# B&R Automation Studio project AutomatedPongGame
Automation Studio 4.12.6.106; technology packages: Acp10Arnc0 5.30.2, mappView 5.16.1

## Configuration AutomatedPongGame_UnitTests

CPU 4PPC70.0573-20B, AutomationRuntime R4.93, Build 4.1.2

### Task classes (Cpu.sw)
```
Cyclic#4 (cycle 10000 us):
  Tests_Incl <- UnitTests.UnitTests.Tests_InclinoSensor_C.prg
  Tests_Padd <- UnitTests.UnitTests.Tests_PaddleMotor_C.prg
  Tests_Fiel <- UnitTests.UnitTests.Tests_FieldMotor_C.prg
  Tests_Pong <- UnitTests.UnitTests.Tests_PongGame_C.prg
  Tests_Ball <- UnitTests.UnitTests.Tests_BallControl_C.prg
  Tests_Fie1 <- UnitTests.UnitTests.Tests_FieldControl_C.prg
  Tests_Dist <- UnitTests.UnitTests.Tests_DistanceSensor_C.prg
  Tests_Shoo <- UnitTests.UnitTests.Tests_Shooter_C.prg
Binaries: mvLoader, udbdef, TCData, iomap, asfw, arconfig, ashwd, sysconf, ashwac
Libraries: Runtime, sys_lib, AsIecCon, astime, AsARCfg, AsBrStr, UnitTest, UtWs, UtMgr, Library, arssl, fileio, standard
```

### Hardware
```
4PPC70_0573_20B : 4PPC70.0573-20B v1.6.1.0
  Connector IF2:
    ActivateDevice = 1
    InaPort = 11160
  ConfigurationID = AutomatedPongGame_TS_UnitTest_Sample
  Cyclic4Duration = 10000
  FileDevice1
  FileDeviceName1 = USER
  FileDevicePath1 = USER_PATH
  ActivateDtmServer = 1
  ActivateOpcUa = 1
  OpcUaInformationModels_PV_Version = 1
  KeyMappingFile = VC\4PPC70_0573_20B.dis
```

## Configuration AutomatedPongGame_config

CPU 4PPC70.0573-20B, AutomationRuntime R4.93, Build 4.1.2, Safety 0.0, Vc V4.73.4

### Task classes (Cpu.sw)
```
Cyclic#1 (cycle 2000 us, tolerance 0 us):
  gAxis01Bas <- gAxis01obj.gAxis01Basic.prg
  gAxis02Bas <- gAxis02obj.gAxis02Basic.prg
  Main <- Main.prg
NcDataObjects: acp10etxen <- acp10etxen.dob, gAxis01a <- gAxis01obj.gAxis01a.dob, gAxis01i <- gAxis01obj.gAxis01i.dob, gAxis02a <- gAxis02obj.gAxis02a.dob, gAxis02i <- gAxis02obj.gAxis02i.dob
VcDataObjects: Visu <- Visu.dob
Binaries: udbdef, FWRules, TCData, mvLoader, vcctext, arialbd, vcpdi855, vcdsloc, vcbclass, vcfntttf, Visu03, vcshared, vcrt, vcpk, vcfile, vccbtn, vcmgr, vctcal, vcptelo, vcalarm, vccnum, vcpdsw, Visu01, vcgclass, vcpdihd, vcpdi815, vcpfppc7, vcdsint, Visu02, calibrib, vccbmp, arial, vccstr, Acp10map, acp10cfg, iomap, ashwac, Role, sysconf, arconfig, asfw, User, ashwd, asnxdb1, User_1
Libraries: standard, sys_lib, brsystem, runtime, AsBrStr, Acp10man, Acp10par, NcGlobal, Acp10sdc, Acp10_MC, Library, arssl, astime, powerlnk, fileio, vcresman, AsARCfg, DataObj
```

### Hardware
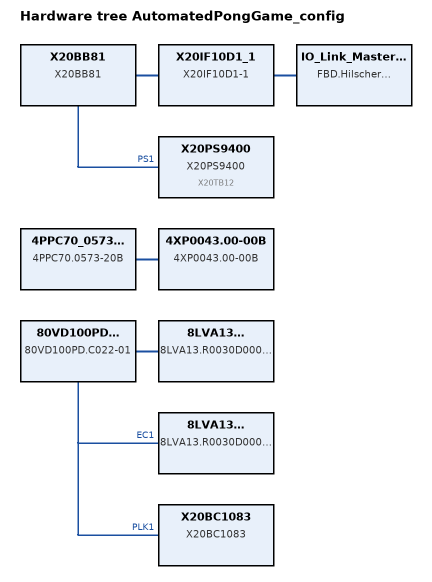
```
4PPC70_0573_20B : 4PPC70.0573-20B v1.6.1.0
  Connector IF1:
    InternetAddress = 192.168.30.1
    SubnetMask = 255.255.255.0
    ActivateIna = 1
  Connector IF2:
    ActivateDevice = 1
    Mode = Manual
    InternetAddress = 192.168.1.20
    SubnetMask = 255.255.255.0
    InaNodeNumber = 0
    Vnc1
    VncAuthentication1 = 1
    VncPasswordViewOnly1 = user
    VncPasswordViewControl1 = admin
    ActivateSnmp = 2
  ConfigurationID = AutomatedPongGame_Config1
  PermanentPvSize = 108
  RemanentGlobalPvSize = 108
  TimerDeviceType = EPLX2X
  TimerDevice = 4PPC70_0573_20B.IF1
  TaskClassIdleTime = 2000
  Cyclic1Duration = 2000
  Cyclic1Tolerance = 0
  Cyclic1Output = 1
  FileDevice1
  FileDeviceName1 = USER
  FileDevicePath1 = USER_PATH
  ActivateDtmServer = 1
  ActivateOpcUa = 1
  OpcUaInformationModels_PV_Version = 1
  VcObjectName = Visu
  KeyMappingFile = VC\4PPC70_0573_20B.dis
4XP0043.00-00B : 4XP0043.00-00B v2.1.1.0  [X2X1 -> 4PPC70_0573_20B.IF5 [Cable Type=X2XCable, Length=10, Version=1.0.0.3]]
80VD100PD.C022-01 : 80VD100PD.C022-01 v2.5.0.0  [PLK1 -> X20BC1083.PLK1 (NodeNumber=2) [Cable Type=PowerlinkCable, Length=10, Version=1.0.0.3]; EC1 -> 8LVA13.R0030D000-0a.EC; EC2 -> 8LVA13.R0030D000-0.EC; MT2 -> 8LVA13.R0030D000-0.MT]
  MotionTP = Acp10Arnc0
  BothEndSwitchesAreNormallyOpen_r1 = on
  QuickStopIsNormallyOpen_r1 = on
  BothEndSwitchesAreNormallyOpen_r2 = on
  QuickStopIsNormallyOpen_r2 = on
8LVA13.R0030D000-0 : 8LVA13.R0030D000-0 v2.2.0.5  [EC -> 80VD100PD.C022-01.EC2; MT -> 80VD100PD.C022-01.MT2]
8LVA13.R0030D000-0a : 8LVA13.R0030D000-0 v2.2.0.5  [EC -> 80VD100PD.C022-01.EC1; MT -> 80VD100PD.C022-01.MT1]
IO_Link_Master_SL_EIP_8P_IP67_V1_5 : FBD.Hilscher.EIGenEDSAdapterDTM.IO-Link Master SL EIP 8P IP67 V1.5 v1.5 (OrderNumber=IO-Link Master SL EIP 8P IP67 V1.5, VendorAddress=192.168.1.150)  [EIP1 -> X20IF10D1_1.IF1]
  DtmId = cae6d7b0-cfd8-47f1-9e8e-3783e9b887dc
  ChannelBlocks_78e66418-9731-44dc-bd45-61a937da4e16  // Module 0
  IO_InputImage_78e66418-9731-44dc-bd45-61a937da4e16  // 446 Byte(s)
  IO_OutputImage_78e66418-9731-44dc-bd45-61a937da4e16  // 302 Byte(s)
X20BB81 : X20BB81 v1.2.0.0
X20BC1083 : X20BC1083 v2.17.0.0  [PLK1 -> 80VD100PD.C022-01.PLK1 (NodeNumber=1) [Cable Type=PowerlinkCable, Length=10, Version=1.0.0.3]; PLK2 -> 4PPC70_0573_20B.IF1 (NodeNumber=1) [Cable Type=PowerlinkCable, Length=10, Version=1.0.0.3]; SL -> X20BB81.SL1]
X20IF10D1_1 : X20IF10D1-1 v1.7.0.0  [SS -> X20BB81.SS1]
  Connector IF1:
    DtmId = 66a43618-f239-4c0c-80e6-69720443d023
  ConfigFile = X20IF10D1_1.dtm
  ConfigModule = asnxdb1
  CycleTime = 2000
X20PS9400 : X20PS9400 v1.9.0.0  [SS1 -> X20TB12.SS; PS -> X20BB81.PS1]
X20TB12 : X20TB12 v1.0.0.0
```

### IoMap.iom - 4PPC70_0573_20B/IoMap.iom
```iecst
VAR_CONFIG
	::digitalInput AT %IB."IO_Link_Master_SL_EIP_8P_IP67_V1_5".Module_0_Input001;
	::gAxis01Bas:BasicControl.Command.MoveJogNeg AT %QX."4XP0043.00-00B".DigitalOutput03;
	::g_Shooter.IO.Shoot AT %QX."4XP0043.00-00B".DigitalOutput07;
	::digitalOutput AT %QB."IO_Link_Master_SL_EIP_8P_IP67_V1_5".Module_0_Output001;
	::g_PaddleMotor.HMI.MoveJogNeg AT %IX."4XP0043.00-00B".DigitalInput01;
	::g_Shooter.HMI.Shoot AT %IX."4XP0043.00-00B".DigitalInput02;
	::g_PaddleMotor.HMI.MoveJogPos AT %IX."4XP0043.00-00B".DigitalInput03;
	::g_DistanceSensorLeft.IO.DataMSB AT %IB."IO_Link_Master_SL_EIP_8P_IP67_V1_5".Module_0_Input415;
	::g_DistanceSensorLeft.IO.DataLSB AT %IB."IO_Link_Master_SL_EIP_8P_IP67_V1_5".Module_0_Input416;
	::g_DistanceSensorRight.IO.DataMSB AT %IB."IO_Link_Master_SL_EIP_8P_IP67_V1_5".Module_0_Input383;
	::g_DistanceSensorRight.IO.DataLSB AT %IB."IO_Link_Master_SL_EIP_8P_IP67_V1_5".Module_0_Input384;
	::g_DistanceSensorMiddle.IO.DataMSB AT %IB."IO_Link_Master_SL_EIP_8P_IP67_V1_5".Module_0_Input351;
	::g_DistanceSensorMiddle.IO.DataLSB AT %IB."IO_Link_Master_SL_EIP_8P_IP67_V1_5".Module_0_Input352;
	::gAxis01Bas:BasicControl.Command.MoveJogPos AT %QX."4XP0043.00-00B".DigitalOutput11;
	::g_InclinoSensor.IO.DataMSB AT %IB."IO_Link_Master_SL_EIP_8P_IP67_V1_5".Module_0_Input319;
	::g_InclinoSensor.IO.DataLSB AT %IB."IO_Link_Master_SL_EIP_8P_IP67_V1_5".Module_0_Input320;
	::g_DistanceSensorMiddle.IO.SensorInfo AT %IB."IO_Link_Master_SL_EIP_8P_IP67_V1_5".Module_0_Input358;
	::g_DistanceSensorRight.IO.SensorInfo AT %IB."IO_Link_Master_SL_EIP_8P_IP67_V1_5".Module_0_Input390;
	::g_DistanceSensorLeft.IO.SensorInfo AT %IB."IO_Link_Master_SL_EIP_8P_IP67_V1_5".Module_0_Input422;
	::g_InclinoSensor.IO.SetCenterPoint AT %QB."IO_Link_Master_SL_EIP_8P_IP67_V1_5".Module_0_Output175;
END_VAR
```

## Configuration Config1

CPU 4PPC70.0573-20B, AutomationRuntime R4.93, Build 4.1.2, Safety 0.0, Vc V4.73.4

### Task classes (Cpu.sw)
```
Cyclic#1 (cycle 2000 us, tolerance 0 us):
  gAxis01Bas <- gAxis01obj.gAxis01Basic.prg
  gAxis02Bas <- gAxis02obj.gAxis02Basic.prg
  Main <- Main.prg
Cyclic#4:
  TonTimer <- Timer_CPP.TonTimer.prg
NcDataObjects: acp10etxen <- acp10etxen.dob, gAxis01a <- gAxis01obj.gAxis01a.dob, gAxis01i <- gAxis01obj.gAxis01i.dob, gAxis02a <- gAxis02obj.gAxis02a.dob, gAxis02i <- gAxis02obj.gAxis02i.dob
VcDataObjects: Visu <- Visu.dob
Binaries: udbdef, FWRules, TCData, mvLoader, vcctext, arialbd, vcpdi855, vcdsloc, vcbclass, vcfntttf, Visu03, vcshared, vcrt, vcpk, vcfile, vccbtn, vcmgr, vctcal, vcptelo, vcalarm, vccnum, vcpdsw, Visu01, vcgclass, vcpdihd, vcpdi815, vcpfppc7, vcdsint, Visu02, calibrib, vccbmp, arial, vccstr, Acp10map, acp10cfg, iomap, ashwac, Role, sysconf, arconfig, asfw, User, ashwd, asnxdb1, User_1
Libraries: Timer, standard, sys_lib, brsystem, runtime, AsBrStr, Acp10man, Acp10par, NcGlobal, Acp10sdc, Acp10_MC, Library, arssl, astime, powerlnk, fileio, dataobj, vcresman
```

### Hardware
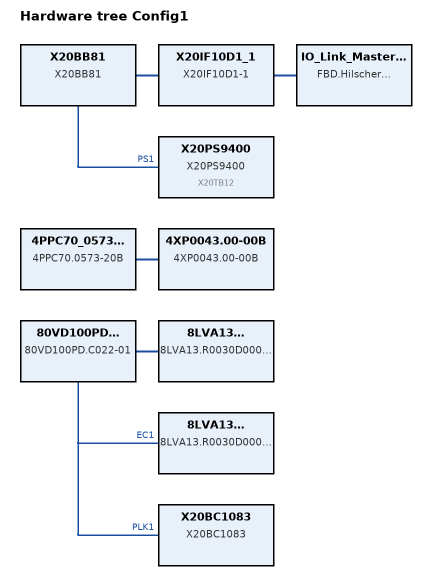
```
4PPC70_0573_20B : 4PPC70.0573-20B v1.6.1.0
  Connector IF1:
    InternetAddress = 192.168.30.1
    SubnetMask = 255.255.255.0
    ActivateIna = 1
  Connector IF2:
    ActivateDevice = 1
    Mode = Manual
    InternetAddress = 192.168.1.20
    SubnetMask = 255.255.255.0
    InaNodeNumber = 0
    Vnc1
    VncAuthentication1 = 1
    VncPasswordViewOnly1 = user
    VncPasswordViewControl1 = admin
    ActivateSnmp = 2
  ConfigurationID = AutomatedPongGame_Config1
  TimerDeviceType = EPLX2X
  TimerDevice = 4PPC70_0573_20B.IF1
  TaskClassIdleTime = 2000
  Cyclic1Duration = 2000
  Cyclic1Tolerance = 0
  Cyclic1Output = 1
  FileDevice1
  FileDeviceName1 = USER
  FileDevicePath1 = USER_PATH
  ActivateDtmServer = 1
  ActivateOpcUa = 1
  OpcUaInformationModels_PV_Version = 1
  VcObjectName = Visu
  KeyMappingFile = VC\4PPC70_0573_20B.dis
4XP0043.00-00B : 4XP0043.00-00B v2.1.1.0  [X2X1 -> 4PPC70_0573_20B.IF5 [Cable Type=X2XCable, Length=10, Version=1.0.0.3]]
80VD100PD.C022-01 : 80VD100PD.C022-01 v2.5.0.0  [PLK1 -> X20BC1083.PLK1 (NodeNumber=2) [Cable Type=PowerlinkCable, Length=10, Version=1.0.0.3]; EC1 -> 8LVA13.R0030D000-0a.EC; EC2 -> 8LVA13.R0030D000-0.EC; MT2 -> 8LVA13.R0030D000-0.MT]
  MotionTP = Acp10Arnc0
  BothEndSwitchesAreNormallyOpen_r1 = on
  QuickStopIsNormallyOpen_r1 = on
  BothEndSwitchesAreNormallyOpen_r2 = on
  QuickStopIsNormallyOpen_r2 = on
8LVA13.R0030D000-0 : 8LVA13.R0030D000-0 v2.2.0.5  [EC -> 80VD100PD.C022-01.EC2; MT -> 80VD100PD.C022-01.MT2]
8LVA13.R0030D000-0a : 8LVA13.R0030D000-0 v2.2.0.5  [EC -> 80VD100PD.C022-01.EC1; MT -> 80VD100PD.C022-01.MT1]
IO_Link_Master_SL_EIP_8P_IP67_V1_5 : FBD.Hilscher.EIGenEDSAdapterDTM.IO-Link Master SL EIP 8P IP67 V1.5 v1.5 (OrderNumber=IO-Link Master SL EIP 8P IP67 V1.5, VendorAddress=192.168.1.150)  [EIP1 -> X20IF10D1_1.IF1]
  DtmId = cae6d7b0-cfd8-47f1-9e8e-3783e9b887dc
  ChannelBlocks_78e66418-9731-44dc-bd45-61a937da4e16  // Module 0
  IO_InputImage_78e66418-9731-44dc-bd45-61a937da4e16  // 446 Byte(s)
  IO_OutputImage_78e66418-9731-44dc-bd45-61a937da4e16  // 302 Byte(s)
X20BB81 : X20BB81 v1.2.0.0
X20BC1083 : X20BC1083 v2.17.0.0  [PLK1 -> 80VD100PD.C022-01.PLK1 (NodeNumber=1) [Cable Type=PowerlinkCable, Length=10, Version=1.0.0.3]; PLK2 -> 4PPC70_0573_20B.IF1 (NodeNumber=1) [Cable Type=PowerlinkCable, Length=10, Version=1.0.0.3]; SL -> X20BB81.SL1]
X20IF10D1_1 : X20IF10D1-1 v1.7.0.0  [SS -> X20BB81.SS1]
  Connector IF1:
    DtmId = 66a43618-f239-4c0c-80e6-69720443d023
  ConfigFile = X20IF10D1_1.dtm
  ConfigModule = asnxdb1
  CycleTime = 2000
X20PS9400 : X20PS9400 v1.9.0.0  [SS1 -> X20TB12.SS; PS -> X20BB81.PS1]
X20TB12 : X20TB12 v1.0.0.0
```

### IoMap.iom - 4PPC70_0573_20B/IoMap.iom
```iecst
VAR_CONFIG
	::digitalInput AT %IB."IO_Link_Master_SL_EIP_8P_IP67_V1_5".Module_0_Input001;
	::gAxis01Bas:BasicControl.Command.MoveJogNeg AT %QX."4XP0043.00-00B".DigitalOutput03;
	::g_Shooter.IO.Shoot AT %QX."4XP0043.00-00B".DigitalOutput07;
	::digitalOutput AT %QB."IO_Link_Master_SL_EIP_8P_IP67_V1_5".Module_0_Output001;
	::g_PaddleMotor.HMI.MoveJogNeg AT %IX."4XP0043.00-00B".DigitalInput01;
	::g_Shooter.HMI.Shoot AT %IX."4XP0043.00-00B".DigitalInput02;
	::g_PaddleMotor.HMI.MoveJogPos AT %IX."4XP0043.00-00B".DigitalInput03;
	::g_DistanceSensorLeft.IO.DataMSB AT %IB."IO_Link_Master_SL_EIP_8P_IP67_V1_5".Module_0_Input415;
	::g_DistanceSensorLeft.IO.DataLSB AT %IB."IO_Link_Master_SL_EIP_8P_IP67_V1_5".Module_0_Input416;
	::g_DistanceSensorRight.IO.DataMSB AT %IB."IO_Link_Master_SL_EIP_8P_IP67_V1_5".Module_0_Input383;
	::g_DistanceSensorRight.IO.DataLSB AT %IB."IO_Link_Master_SL_EIP_8P_IP67_V1_5".Module_0_Input384;
	::g_DistanceSensorMiddle.IO.DataMSB AT %IB."IO_Link_Master_SL_EIP_8P_IP67_V1_5".Module_0_Input351;
	::g_DistanceSensorMiddle.IO.DataLSB AT %IB."IO_Link_Master_SL_EIP_8P_IP67_V1_5".Module_0_Input352;
	::gAxis01Bas:BasicControl.Command.MoveJogPos AT %QX."4XP0043.00-00B".DigitalOutput11;
	::g_InclinoSensor.IO.DataMSB AT %IB."IO_Link_Master_SL_EIP_8P_IP67_V1_5".Module_0_Input319;
	::g_InclinoSensor.IO.DataLSB AT %IB."IO_Link_Master_SL_EIP_8P_IP67_V1_5".Module_0_Input320;
	::g_DistanceSensorMiddle.IO.SensorInfo AT %IB."IO_Link_Master_SL_EIP_8P_IP67_V1_5".Module_0_Input358;
	::g_DistanceSensorRight.IO.SensorInfo AT %IB."IO_Link_Master_SL_EIP_8P_IP67_V1_5".Module_0_Input390;
	::g_DistanceSensorLeft.IO.SensorInfo AT %IB."IO_Link_Master_SL_EIP_8P_IP67_V1_5".Module_0_Input422;
END_VAR
```

### Acp10cfg.ncc - 4PPC70_0573_20B/Motion/Acp10cfg.ncc
```
NcConfiguration (Version=5.30.2, NcSwId=Acp10)
  ACP10CF1_typ:
    cnt_nettrc_rec_drive = 1500
    bufsize_trace_upload = 1200
    tc_nc_man_task = Cyclic #1
    glob_pv_as_ncobject = Yes
    ncsys_dl_broadcast = Yes
    ncsys_dl_acp_reset = Yes
    safemc_log_err_to_ax = Yes
    network_init:
      ncsw_init_execute = Yes
      automatic_execute = No
      node_nr_warning = Yes
      net_err_before_ncact = Yes
    nettrc:
      enter_parsecrec = Yes
      enter_ncaction = Yes
      save_ring_startidx = Yes
    cam_prof_download:
      cam_dat_dl_parallel = No
      tc_cam_dl_parallel = Task class for NC Manager task
    plk_if[0]:
      if_name = IF1
      tc_CycDat_PLCopen = Task class for NC Manager task
      mc_broadcast_extdat = No
```

### Acp10map.ncm - 4PPC70_0573_20B/Motion/Acp10map.ncm
```
NcMapping (NcSwId=Acp10)
  NcObject gAxis01 (ModuleId=80VD100PD.C022-01, Type=ncAXIS, Channel=1, AcoposSimulation=Off, InitParameter=gAxis01i, AcoposParameter=gAxis01a, Disabled=FALSE, ModuleDisabled=FALSE)
  NcObject gAxis02 (ModuleId=80VD100PD.C022-01, Type=ncAXIS, Channel=2, AcoposSimulation=Off, InitParameter=gAxis02i, AcoposParameter=gAxis02a, Disabled=FALSE, ModuleDisabled=FALSE)
  NcObject 80VD100PD.C022-01_ncV_AXIS1 (ModuleId=80VD100PD.C022-01, Type=ncV_AXIS, Channel=1, Disabled=TRUE, ModuleDisabled=FALSE)
  NcObject 80VD100PD.C022-01_ncV_AXIS2 (ModuleId=80VD100PD.C022-01, Type=ncV_AXIS, Channel=2, Disabled=TRUE, ModuleDisabled=FALSE)
```

## Configuration TS_UnitTest_Sample

### Task classes (Cpu.sw)
```
Cyclic#4 (cycle 10000 us):
  SPL_CalcTe <- UnitTestSample.Samples.Tests_Program.Tests_MyCalcLib_C.SPL_CalcTest.prg
  SPL_CalcT1 <- UnitTestSample.Samples.Tests_Program.Tests_MyCalcLib_C.SPL_CalcTest_Variants.prg
  Tests_Padd <- UnitTests.HelperTool_Supported.Tests_PaddleMotor_C.prg
Binaries: mvLoader, udbdef, TCData, iomap, asfw, arconfig, ashwd, sysconf, ashwac
Libraries: Runtime, sys_lib, AsIecCon, astime, AsARCfg, AsBrStr, UnitTest, UtWs, UtMgr, SPLMyCalc, Library, arssl, fileio
```

### Hardware
```
4PPC70_0573_20B : 4PPC70.0573-20B v1.6.1.0
  Connector IF2:
    ActivateDevice = 1
    InaPort = 11160
  ConfigurationID = AutomatedPongGame_TS_UnitTest_Sample
  Cyclic4Duration = 10000
  FileDevice1
  FileDeviceName1 = USER
  FileDevicePath1 = USER_PATH
  KeyMappingFile = VC\4PPC70_0573_20B.dis
```

## Logical view

Binary libraries used (declarations not repeated): UtMgr 2.02.0, UtWs 2.02.0, operator, runtime, astime, AsIecCon, standard, sys_lib, brsystem, AsBrStr, Acp10man 5.30.2, Acp10par 5.30.2, NcGlobal 5.30.2, Acp10sdc 5.30.2, Acp10_MC 5.30.2, AsARCfg, DataObj

### Global.var - Global variables
```iecst
VAR
	gAxis01 : ACP10AXIS_typ;
	gAxis02 : ACP10AXIS_typ;
	digitalInput : USINT;
	g_PongGame : UDT_PongGame := (ALM:=(PaddleAxisError:=FALSE,ShooterError:=FALSE,TiltAxisError:=FALSE),CS:=(AutoMode:=FALSE,ErrorAcknowledge:=FALSE,Initialize:=FALSE,Start:=FALSE,StopGame:=FALSE),HMI:=(AutoMode:=FALSE,ErrorAcknowledge:=FALSE,Initialize:=FALSE,Start:=FALSE,StopGame:=FALSE),PAR:=(Score:=0),STS:=(Disabled:=TRUE,AlarmActive:=FALSE,Idle:=FALSE,Initializing:=FALSE,Running:=FALSE,StateInt:=0,AutoActive:=FALSE,Interlocked:=FALSE));
	g_BallControl : UDT_BallControl := (ALM:=(ShooterAlarm:=FALSE,MotorAlarm:=FALSE,DistanceSensorAlarm:=FALSE),CS:=(AutoMode:=FALSE,Initialize:=FALSE,Shoot:=FALSE,Start:=FALSE,Stop:=FALSE,Interlock:=FALSE,ChangePosition:=FALSE,ErrorAcknowledge:=FALSE,StopGame:=FALSE),HMI:=(dummy:=FALSE),PAR:=(Position:=0),STS:=(Disabled:=TRUE,Idle:=FALSE,AlarmActive:=FALSE,Initializing:=FALSE,Running:=FALSE,Interlocked:=FALSE,StateInt:=0,AutoActive:=FALSE));
	g_FieldControl : UDT_FieldControl := (ALM:=(MotorAlarm:=FALSE),CS:=(MoveToAngle:=FALSE,Initialize:=FALSE,Stop:=FALSE,StopGame:=FALSE,Start:=FALSE,ErrorAcknowledge:=FALSE,Interlock:=FALSE,SetCenterPoint:=FALSE),HMI:=(IncreaseAngle:=FALSE,DecreaseAngle:=FALSE),PAR:=(Angle:=3),STS:=(Disabled:=TRUE,Idle:=FALSE,Running:=FALSE,AlarmActive:=FALSE,Initializing:=FALSE,Moving:=FALSE,StateInt:=0,Interlocked:=FALSE,AutoActive:=FALSE,AtTargetPosition:=FALSE));
	g_DistanceSensorLeft : UDT_DistanceSensor := (ALM:=(OutOfBounds:=FALSE),CS:=(Power:=TRUE),HMI:=(Power:=FALSE),PAR:=(dummy:=0),STS:=(TooClose:=FALSE,TooFar:=FALSE,StateInt:=0,AlarmActive:=FALSE));
	g_PaddleMotor : UDT_PaddleMotor := (ALM:=(MotorError:=FALSE,ErrorID:=0),CS:=(Home:=FALSE,MoveAbsolute:=FALSE,MoveJogNeg:=FALSE,MoveJogPos:=FALSE,Power:=FALSE,Stop:=FALSE,ErrorAcknowledge:=FALSE,Start:=FALSE,Interlock:=FALSE,AutoMode:=FALSE,Initialize:=FALSE,StopGame:=FALSE),HMI:=(Home:=FALSE,MoveAbsolute:=FALSE,MoveJogNeg:=FALSE,MoveJogPos:=FALSE,Power:=FALSE,Stop:=FALSE,Start:=FALSE,IncreaseJogSpeed:=FALSE,DecreaseJogSpeed:=FALSE,ErrorAcknowledge:=FALSE,IncreaseAccDec:=FALSE,DecreaseAccDec:=FALSE,Initialize:=FALSE),IO:=(EndButton:=FALSE,Power:=TRUE,Home:=TRUE,ErrorAcknowledge:=FALSE,MoveJogNeg:=FALSE,MoveJogPos:=FALSE,Stop:=FALSE,MoveAbsolute:=FALSE,Acceleration:=40000,Deceleration:=40000,JogVelocity:=400,Velocity:=400,Position:=0),PAR:=(Acceleration:=40000,Deceleration:=40000,JogVelocity:=1000,Velocity:=1000,Position:=0),STS:=(Disabled:=TRUE,Initializing:=FALSE,Idle:=FALSE,AlarmActive:=FALSE,Moving:=FALSE,StandStill:=TRUE,AtTargetPosition:=FALSE,ActPosition:=0,Interlocked:=FALSE,PowerOn:=FALSE,AutoActive:=FALSE,StateInt:=0,ActVelocity:=0,EndButtonHit:=FALSE));
	g_FieldMotor : UDT_FieldMotor := (ALM:=(MotorError:=FALSE,ErrorID:=0),CS:=(Home:=FALSE,MoveAbsolute:=FALSE,MoveJogNeg:=FALSE,MoveJogPos:=FALSE,Power:=FALSE,Stop:=FALSE,StopGame:=FALSE,ErrorAcknowledge:=FALSE,Start:=FALSE,Interlock:=FALSE,Initialize:=FALSE,SetCenterPoint:=FALSE),HMI:=(MoveAbsolute:=FALSE,MoveJogNeg:=FALSE,MoveJogPos:=FALSE,Power:=FALSE,IncreaseJogSpeed:=FALSE,DecreaseJogSpeed:=FALSE,ErrorAcknowledge:=FALSE),IO:=(EndButton:=FALSE,Power:=TRUE,Home:=TRUE,ErrorAcknowledge:=FALSE,MoveJogNeg:=FALSE,MoveJogPos:=FALSE,Stop:=FALSE,MoveAbsolute:=FALSE,Acceleration:=40000,Deceleration:=40000,JogVelocity:=400,Velocity:=400,Position:=0),PAR:=(Acceleration:=40000,Deceleration:=40000,JogVelocity:=1000,Velocity:=1000,Position:=0),STS:=(Disabled:=TRUE,Initializing:=FALSE,Idle:=FALSE,Running:=FALSE,AlarmActive:=FALSE,Moving:=FALSE,StandStill:=TRUE,AtTargetPosition:=FALSE,ActPosition:=0,Interlocked:=FALSE,PowerOn:=FALSE,AutoActive:=FALSE,StateInt:=0,ActVelocity:=0,EndButtonHit:=FALSE,TimerStarted:=FALSE,TimerEnded:=FALSE));
	g_InclinoSensor : UDT_InclinoSensor := (CS:=(Power:=TRUE,Reset:=FALSE),HMI:=(Power:=FALSE,Reset:=FALSE),STS:=(PowerOn:=TRUE));
	digitalOutput : USINT;
	g_Shooter : UDT_Shooter := (CS:=(Interlock:=FALSE,EnableFan:=FALSE,Shoot:=FALSE),HMI:=(EnableFan:=FALSE,Shoot:=FALSE,IncreaseIntensity:=FALSE,DecreaseIntensity:=FALSE),IO:=(EnableFan:=FALSE,Shoot:=FALSE),STS:=(Disabled:=TRUE,Idle:=FALSE,Interlocked:=FALSE,AlarmActive:=FALSE,AutoActive:=FALSE,Shooting:=FALSE,StateInt:=0));
	g_DistanceSensorRight : UDT_DistanceSensor := (ALM:=(OutOfBounds:=FALSE),CS:=(Power:=TRUE),HMI:=(Power:=FALSE),STS:=(PowerOn:=TRUE,StateInt:=0,AlarmActive:=FALSE));
	g_DistanceSensorMiddle : UDT_DistanceSensor := (ALM:=(OutOfBounds:=FALSE),CS:=(Power:=TRUE),HMI:=(Power:=FALSE));
END_VAR
```

### Package Logical/Libraries - Global libraries

### Library Logical/Libraries/UnitTest/UnitTest (ANSIC, version 2.02.0) - Static library for UnitTest programs written in ANSI C /C++

#### UnitTest.h
```c
/*****************************************************************************
 * COPYRIGHT (C) BERNECKER + RAINER
 *****************************************************************************
 * Library:  UnitTest
 * File:     UnitTest.h
 * Author:   B+R
 *****************************************************************************
 * Description: Static library for UnitTest programs written in ANSI C /C++
 *
 * Add the path "\Logical\TS_UnitTest\Libraries\UnitTest\" to the
 * "Additional include directories" in the tab "Build" (PLC Properties)
 ******************************************************************************/

#ifndef	__UNITTEST_H__
#define	__UNITTEST_H__
#ifdef __cplusplus
extern "C"
{
#endif
#include <bur/plctypes.h>

#ifndef NULL
#define	NULL	0
#endif
#include "include/Test.h"

#include "include/TestCase.h"
#include "include/TestListener.h"
#include "include/TestResult.h"
#include "include/TestCaller.h"

#include "include/AssertImpl.h"
#include "include/HelperMacro.h"
#include "include/utRunner.h"

/* function is a test case */
#define _TEST 			static testStatusEnum

/* function is a setup */
#define _SETUP_TEST 	static testStatusEnum 	setupTest

/* function is a teardown */
#define _TEARDOWN_TEST 	static testStatusEnum 	teardownTest

/* function is a setup for whole test set */
#define _SETUP_SET		static testStatusEnum	setupSet

/* function is a teardown for whole test set */
#define _TEARDOWN_SET 	static testStatusEnum	teardownSet

/* function is a cyclic handler for test set */
#define _CYCLIC_SET		static void 			cyclicSetCaller

/* Skipped test case */
#define SKIP_TEST  		_TEST
/* Skip all test cases of set */
#define SKIP_TEST_SET

/* Dummies for smart edit autocompletion.
See AssertImpl.h for real macros used by the compiler  */
#ifdef _SMART_EDIT_DUMMY_

/* String comparison.
Returns true if the strings are equal. */
BOOL TEST_ASSERT_EQUAL_STRING(char *expected,char  *actual);
/* Wstring comparison.
Returns true if the WSTRINGS are equal. */
BOOL TEST_ASSERT_EQUAL_WSTRING(unsigned short *expected,unsigned short *actual);
 /* Compares two memory blocks.
Returns true if [size] bytes are equal. */
BOOL TEST_ASSERT_EQUAL_MEM(void *expected, void *actual,UDINT size);
/* Compares integer values. Usable for all integer types.
Avoid comparison of unsigned with signed types.
Returns true if they are equal.
Note: If different, values are reported as DINT values in the test report */
BOOL TEST_ASSERT_EQUAL_INT(expected, actual);

/* Compares REAL values with delta = (expected * TEST_FLOAT_PRECISION).
Returns true if (difference <= delta) */
BOOL TEST_ASSERT_EQUAL_REAL(REAL expected,REAL actual);
/* Compares REAL values with explicit delta.
Returns true if (difference <= delta) */
BOOL TEST_ASSERT_REAL_WITHIN(REAL delta, REAL expected, REAL actual);
/* Compares LREAL values with delta = (expected * TEST_DOUBLE_PRECISION).
Returns true if (difference <= delta) */
BOOL TEST_ASSERT_EQUAL_LREAL(LREAL expected,LREAL  actual);
/* Compares LREAL values with explicit delta.
Returns true if (difference <= delta) */
BOOL TEST_ASSERT_LREAL_WITHIN(LREAL delta, LREAL expected, LREAL actual);

/* Compares float values with delta = (expected * TEST_FLOAT_PRECISION).
Returns true if (difference <= delta) */
BOOL TEST_ASSERT_EQUAL_FLOAT(float expected, float actual);
/* Compares float values with explicit delta.
Returns true if (difference <= delta) */
BOOL TEST_ASSERT_FLOAT_WITHIN(float delta, float expected, float actual);
/* Compares double values with delta = (expected * TEST_DOUBLE_PRECISION).
Returns true if (difference <= delta) */
BOOL TEST_ASSERT_EQUAL_DOUBLE(double expected, double actual);
/* Compares double values with explicit delta.
Returns true if (difference <= delta) */
BOOL TEST_ASSERT_DOUBLE_WITHIN(double delta, double expected, double actual);

/* Returns true if pointer is null */
BOOL TEST_ASSERT_NULL(void *pointer);
/* Returns true if pointer is not null */
BOOL TEST_ASSERT_NOT_NULL(void *pointer);
/* Returns true, if condition evals to  true */
BOOL TEST_ASSERT_MESSAGE(condition, char *message);
/* Returns true, if condition evals to  true */
BOOL TEST_ASSERT(condition);

/* Returns always false */
BOOL TEST_FAIL(char *message);

/* Add a note to the test report */
void TEST_INFO(char *message);
/* Add a note with location information to the test report */
void TEST_INFO_POS(char *message);

#ifdef __cplusplus
/* Test if expression throws given exception.
Catches all other exceptions as failure.
Note: Available for C++ only */
void TEST_ASSERT_THROW(expression, type);

/* Fails if expression throws any exceptions.
Note: Available for C++ only*/
void TEST_ASSERT_NO_THROW(expression);
#endif

/* Adds a test function with description to the Testfixture.
See UNITTEST_FIXTURES() */
void new_TestFixture(char *name, _TEST function);

/* Adds a test function with description to the Testfixture.
This test will be skipped
See UNITTEST_FIXTURES() */
void skipTestFixture(char *name, _TEST function);

/* Defines the order of test cases.
Should look like this
UNITTEST_FIXTURES(fixtures)
{
	new_TestFixture("test_1",test_1),
	new_TestFixture("test_2",test_2),
	new_TestFixture("test_3",test_3)
}
*/
void UNITTEST_FIXTURES(fixtures)

/* Standard UnitTest caller without any setup / teardown methods*/
void UNITTEST_CALLER_TEST(caller, char *name, fixtures);

/* Standard UnitTest caller with macro setup / teardown for tests*/
void UNITTEST_CALLER_BASIC(caller, char *name, fixtures);

/* UnitTest caller with macro setup / teardown for tests and test set */
void UNITTEST_CALLER_SET(caller, char *name, fixtures);

/* UnitTest caller with macro setup / teardown for tests and test set and cylic*/
void UNITTEST_CALLER_COMPLETE(caller, char *name, fixtures);

/* UnitTest caller with explicit setup / teardown for suite */
void UNITTEST_CALLER_SET_EXPLICIT(caller,name,setupTest,teardownTest,fixtures, setupSuite, teardownSuite);

/* UnitTest caller with explicit setup / teardown for suite and cylic */
void UNITTEST_CALLER_COMPLETE_EXPLICIT(caller,name,setupTest,teardownTest,fixtures, setupSuite, teardownSuite, cyclicCaller);

/* Adds a test set with description to the fixture of test sets.
See UNITTEST_TESTSET_FIXTURES() */
void new_TestSet(testcaller);

/* Defines the order of test sets.
Should look like this
UNITTEST_TESTSET_FIXTURES(fixtures)
{
	new_TestSet(testSet_1),
	new_TestSet(testSet_2),
	new_TestSet(testSet_3)
}*/
void UNITTEST_TESTSET_FIXTURES(fixtures);

/* Defines the test set list handling structure*/
void UNTITTEST_TESTSET_HANDLER();

#endif /*_SMART_EDIT_DUMMY_*/

/*
 Use to declare Test set for use in list of test sets of test programm
 See usage in autogeneratedFile.c / FixtureOfTestSets.c
*/
#define UNITTEST_TESTSET_DECLARATION 	extern const TestCaller

/* Default factor for precision used to test if REAL / float values  are equal.
(0.00001f) */
#define TEST_FLOAT_PRECISION 	(0.00001f)
/* Default factor for precision used to test if LREAL / double values  are equal.
(1e - 12f) */
#define TEST_DOUBLE_PRECISION 	(1e-12f)

#if (__GNUC__ != 4) || (__GNUC_MINOR__ != 1) || (__GNUC_PATCHLEVEL__ != 2)
#warning UnitTest is compiled with GCC version 4.1.2. To use UnitTest switch GCC version to 4.1.2 or use different solution package
#endif

#define UNIT_TEST_LIBRARY_VERSION  			"2.02.0"

#ifdef __cplusplus
};
#endif

#include "include/asserts.hpp"

#endif/*__UNITTEST_H__*/
```

### Library Logical/Libraries/Library (ANSIC)

#### UDT.typ
```iecst
TYPE
	UDT_PongGame : 	STRUCT
		ALM : UDT_PongGame_ALM;
		CS : UDT_PongGame_CS;
		HMI : UDT_PongGame_HMI;
		PAR : UDT_PongGame_PAR;
		STS : UDT_PongGame_STS;
	END_STRUCT;
	UDT_FieldControl : 	STRUCT
		ALM : UDT_FieldControl_ALM;
		CS : UDT_FieldControl_CS;
		HMI : UDT_FieldControl_HMI;
		PAR : UDT_FieldControl_PAR;
		STS : UDT_FieldControl_STS;
	END_STRUCT;
	UDT_BallControl : 	STRUCT
		ALM : UDT_BallControl_ALM;
		CS : UDT_BallControl_CS;
		HMI : UDT_BallControl_HMI;
		PAR : UDT_BallControl_PAR;
		STS : UDT_BallControl_STS;
	END_STRUCT;
	UDT_InclinoSensor : 	STRUCT
		ALM : UDT_InclinoSensor_ALM;
		CS : UDT_InclinoSensor_CS;
		HMI : UDT_InclinoSensor_HMI;
		PAR : UDT_InclinoSensor_PAR;
		STS : UDT_InclinoSensor_STS;
		IO : UDT_InclinoSensor_IO;
	END_STRUCT;
	UDT_FieldMotor : 	STRUCT
		ALM : UDT_FieldMotor_ALM;
		CS : UDT_FieldMotor_CS;
		HMI : UDT_FieldMotor_HMI;
		IO : UDT_FieldMotor_IO;
		PAR : UDT_FieldMotor_PAR;
		STS : UDT_FieldMotor_STS;
	END_STRUCT;
	UDT_Shooter : 	STRUCT
		ALM : UDT_Shooter_ALM;
		CS : UDT_Shooter_CS;
		HMI : UDT_Shooter_HMI;
		IO : UDT_Shooter_IO;
		PAR : UDT_Shooter_PAR;
		STS : UDT_Shooter_STS;
	END_STRUCT;
	UDT_DistanceSensor : 	STRUCT
		ALM : UDT_DistanceSensor_ALM;
		CS : UDT_DistanceSensor_CS;
		HMI : UDT_DistanceSensor_HMI;
		IO : UDT_DistanceSensor_IO;
		PAR : UDT_DistanceSensor_PAR;
		STS : UDT_DistanceSensor_STS;
	END_STRUCT;
	UDT_PaddleMotor : 	STRUCT
		ALM : UDT_PaddleMotor_ALM;
		CS : UDT_PaddleMotor_CS;
		HMI : UDT_PaddleMotor_HMI;
		IO : UDT_PaddleMotor_IO;
		PAR : UDT_PaddleMotor_PAR;
		STS : UDT_PaddleMotor_STS;
	END_STRUCT;
END_TYPE
```

#### Library.fun
```iecst
{REDUND_ERROR} FUNCTION_BLOCK FB_PaddleMotor (*TODO: Add your comment here*) (*$GROUP=User,$CAT=User,$GROUPICON=User.png,$CATICON=User.png*)
	VAR_INPUT
		digitalInput : USINT;
	END_VAR
	VAR_IN_OUT
		PaddleMotor : UDT_PaddleMotor;
	END_VAR
END_FUNCTION_BLOCK

{REDUND_ERROR} FUNCTION_BLOCK FB_DistanceSensor (*TODO: Add your comment here*) (*$GROUP=User,$CAT=User,$GROUPICON=User.png,$CATICON=User.png*)
	VAR_IN_OUT
		DistanceSensorLeft : UDT_DistanceSensor;
		DistanceSensorMiddle : UDT_DistanceSensor;
		DistanceSensorRight : UDT_DistanceSensor;
	END_VAR
END_FUNCTION_BLOCK

{REDUND_ERROR} FUNCTION_BLOCK FB_Shooter (*TODO: Add your comment here*) (*$GROUP=User,$CAT=User,$GROUPICON=User.png,$CATICON=User.png*)
	VAR_OUTPUT
		digitalOutput : USINT;
	END_VAR
	VAR_IN_OUT
		Shooter : UDT_Shooter;
	END_VAR
END_FUNCTION_BLOCK

{REDUND_ERROR} FUNCTION_BLOCK FB_FieldMotor (*TODO: Add your comment here*) (*$GROUP=User,$CAT=User,$GROUPICON=User.png,$CATICON=User.png*)
	VAR_INPUT
		digitalInput : USINT;
	END_VAR
	VAR_IN_OUT
		FieldMotor : UDT_FieldMotor;
	END_VAR
END_FUNCTION_BLOCK

{REDUND_ERROR} FUNCTION_BLOCK FB_InclinoSensor (*TODO: Add your comment here*) (*$GROUP=User,$CAT=User,$GROUPICON=User.png,$CATICON=User.png*)
	VAR_IN_OUT
		InclinoSensor : UDT_InclinoSensor;
	END_VAR
END_FUNCTION_BLOCK

{REDUND_ERROR} {REDUND_UNREPLICABLE} FUNCTION_BLOCK FB_BallControl (*TODO: Add your comment here*) (*$GROUP=User,$CAT=User,$GROUPICON=User.png,$CATICON=User.png*)
	VAR_IN_OUT
		BallControl : UDT_BallControl;
		PaddleMotor : UDT_PaddleMotor;
		Shooter : UDT_Shooter;
		DistanceSensorLeft : UDT_DistanceSensor;
		DistanceSensorMiddle : UDT_DistanceSensor;
		DistanceSensorRight : UDT_DistanceSensor;
	END_VAR
END_FUNCTION_BLOCK

{REDUND_ERROR} FUNCTION_BLOCK FB_FieldControl (*TODO: Add your comment here*) (*$GROUP=User,$CAT=User,$GROUPICON=User.png,$CATICON=User.png*)
	VAR_IN_OUT
		FieldMotor : UDT_FieldMotor;
		FieldControl : UDT_FieldControl;
		InclinoSensor : UDT_InclinoSensor;
	END_VAR
END_FUNCTION_BLOCK

{REDUND_ERROR} FUNCTION_BLOCK FB_PongGame (*TODO: Add your comment here*) (*$GROUP=User,$CAT=User,$GROUPICON=User.png,$CATICON=User.png*)
	VAR_IN_OUT
		PongGame : UDT_PongGame;
		BallControl : UDT_BallControl;
		FieldControl : UDT_FieldControl;
	END_VAR
END_FUNCTION_BLOCK
```

#### UDT_DistanceSensor.typ
```iecst
TYPE
	UDT_DistanceSensor_CS : 	STRUCT
		Power : BOOL;
	END_STRUCT;
	UDT_DistanceSensor_HMI : 	STRUCT
		dummy : BOOL;
	END_STRUCT;
	UDT_DistanceSensor_PAR : 	STRUCT
		dummy : USINT;
	END_STRUCT;
	UDT_DistanceSensor_STS : 	STRUCT
		Distance : INT;
		Reflectivity : INT;
		TooClose : BOOL;
		TooFar : BOOL;
		Valid : BOOL;
		DeviceStatus : UINT;
		PowerOn : BOOL;
		StateInt : USINT;
		AlarmActive : BOOL;
		AlarmActiveColour : USINT;
		BallDetected : BOOL;
	END_STRUCT;
	UDT_DistanceSensor_ALM : 	STRUCT
		OutOfBounds : BOOL;
	END_STRUCT;
	UDT_DistanceSensor_IO : 	STRUCT
		OUT1 : BOOL;
		OUT2 : BOOL;
		DataMSB : USINT;
		DataLSB : USINT;
		SensorInfo : USINT; (*bit 0 = OUT1 (1 als <300mm) , bit 1 = OUT2 (1 als <50mm) , bit 4-7 device status*)
	END_STRUCT;
END_TYPE
```

#### UDT_PaddleMotor.typ
```iecst
TYPE
	UDT_PaddleMotor_CS : 	STRUCT
		Home : BOOL;
		MoveAbsolute : BOOL;
		MoveJogNeg : BOOL;
		MoveJogPos : BOOL;
		Power : BOOL;
		Stop : BOOL;
		ErrorAcknowledge : BOOL;
		Start : BOOL;
		Interlock : BOOL;
		AutoMode : BOOL;
		Initialize : BOOL;
		StopGame : BOOL;
	END_STRUCT;
	UDT_PaddleMotor_HMI : 	STRUCT
		MoveAbsolute : BOOL;
		MoveJogNeg : BOOL;
		MoveJogPos : BOOL;
		IncreaseJogSpeed : BOOL;
		DecreaseJogSpeed : BOOL;
		ErrorAcknowledge : BOOL;
	END_STRUCT;
	UDT_PaddleMotor_PAR : 	STRUCT
		Acceleration : REAL;
		Deceleration : REAL;
		JogVelocity : REAL;
		Velocity : REAL;
		Position : REAL;
	END_STRUCT;
	UDT_PaddleMotor_STS : 	STRUCT
		Disabled : BOOL;
		Initializing : BOOL;
		Idle : BOOL;
		Running : BOOL;
		AlarmActive : BOOL;
		Moving : BOOL;
		StandStill : BOOL;
		AtTargetPosition : BOOL;
		ActPosition : REAL;
		ActVelocity : REAL;
		Interlocked : BOOL;
		PowerOn : BOOL;
		AutoActive : BOOL;
		StateInt : USINT;
		EndButtonHit : BOOL;
		TimerStarted : BOOL;
		TimerEnded : BOOL;
		ReferencePosition : REAL;
		ReferenceSet : BOOL;
		AlarmActiveColour : USINT;
	END_STRUCT;
	UDT_PaddleMotor_ALM : 	STRUCT
		MotorError : BOOL;
		ErrorID : UINT;
		ErrorText : ARRAY[0..3]OF STRING[79];
	END_STRUCT;
	UDT_PaddleMotor_IO : 	STRUCT
		EndButton : BOOL;
		Power : BOOL;
		Home : BOOL;
		ErrorAcknowledge : BOOL;
		MoveJogNeg : BOOL;
		MoveJogPos : BOOL;
		Stop : BOOL;
		MoveAbsolute : BOOL;
		Acceleration : REAL;
		Deceleration : REAL;
		JogVelocity : REAL;
		Velocity : REAL;
		Position : REAL;
	END_STRUCT;
END_TYPE
```

#### UDT_PongGame.typ
```iecst
TYPE
	UDT_PongGame_CS : 	STRUCT
		AutoMode : BOOL;
		ErrorAcknowledge : BOOL;
		Initialize : BOOL;
		Start : BOOL;
		StopGame : BOOL;
	END_STRUCT;
	UDT_PongGame_HMI : 	STRUCT
		AutoMode : BOOL;
		ErrorAcknowledge : BOOL;
		Initialize : BOOL;
		Start : BOOL;
		StopGame : BOOL;
	END_STRUCT;
	UDT_PongGame_PAR : 	STRUCT
		Highscore : UINT;
		Score : UINT;
	END_STRUCT;
	UDT_PongGame_STS : 	STRUCT
		Disabled : BOOL;
		AlarmActive : BOOL;
		Idle : BOOL;
		Initializing : BOOL;
		Running : BOOL;
		StateInt : USINT;
		AutoActive : BOOL;
		Interlocked : BOOL;
		AlarmActiveColour : USINT;
		GameStopped : BOOL;
		StateString : STRING[80];
	END_STRUCT;
	UDT_PongGame_ALM : 	STRUCT
		dummy : BOOL;
	END_STRUCT;
END_TYPE
```

#### UDT_FieldControl.typ
```iecst
TYPE
	UDT_FieldControl_CS : 	STRUCT
		MoveToAngle : BOOL;
		Initialize : BOOL;
		Stop : BOOL;
		StopGame : BOOL;
		Start : BOOL;
		ErrorAcknowledge : BOOL;
		Interlock : BOOL;
		SetCenterPoint : BOOL;
	END_STRUCT;
	UDT_FieldControl_HMI : 	STRUCT
		IncreaseAngle : BOOL;
		DecreaseAngle : BOOL;
	END_STRUCT;
	UDT_FieldControl_PAR : 	STRUCT
		Angle : REAL;
	END_STRUCT;
	UDT_FieldControl_STS : 	STRUCT
		Disabled : BOOL;
		Idle : BOOL;
		Running : BOOL;
		AlarmActive : BOOL;
		Initializing : BOOL;
		Moving : BOOL;
		StateInt : USINT;
		Interlocked : BOOL;
		AutoActive : BOOL;
		CurrentAngle : REAL;
		AtTargetPosition : BOOL;
	END_STRUCT;
	UDT_FieldControl_ALM : 	STRUCT
		dummy : BOOL;
	END_STRUCT;
END_TYPE
```

#### UDT_BallControl.typ
```iecst
TYPE
	UDT_BallControl_CS : 	STRUCT
		AutoMode : BOOL;
		Initialize : BOOL;
		Shoot : BOOL;
		Start : BOOL;
		Stop : BOOL;
		Interlock : BOOL;
		ChangePosition : BOOL;
		ErrorAcknowledge : BOOL;
		StopGame : BOOL;
	END_STRUCT;
	UDT_BallControl_HMI : 	STRUCT
		dummy : BOOL;
	END_STRUCT;
	UDT_BallControl_PAR : 	STRUCT
		Position : REAL;
		DesiredPosition : REAL;
	END_STRUCT;
	UDT_BallControl_STS : 	STRUCT
		Disabled : BOOL;
		Idle : BOOL;
		AlarmActive : BOOL;
		Initializing : BOOL;
		Running : BOOL;
		Interlocked : BOOL;
		StateInt : USINT;
		AutoActive : BOOL;
		BallVelocity : REAL;
		ShootState : USINT;
		TimeToPaddleMS : DINT;
		ShootCycleCompleted : BOOL;
		PrevShootState : USINT;
		NewShootCycleTimerET : UINT;
		GameOver : BOOL;
	END_STRUCT;
	UDT_BallControl_ALM : 	STRUCT
		ShooterAlarm : BOOL;
		MotorAlarm : BOOL;
		DistanceSensorAlarm : BOOL;
	END_STRUCT;
END_TYPE
```

#### UDT_InclinoSensor.typ
```iecst
TYPE
	UDT_InclinoSensor_CS : 	STRUCT
		Power : BOOL;
		Reset : BOOL;
		SetCenterPoint : BOOL;
	END_STRUCT;
	UDT_InclinoSensor_HMI : 	STRUCT
		Power : BOOL;
		Reset : BOOL;
	END_STRUCT;
	UDT_InclinoSensor_PAR : 	STRUCT
		dummy : USINT;
	END_STRUCT;
	UDT_InclinoSensor_STS : 	STRUCT
		CurrentAngle : REAL;
		PowerOn : BOOL;
		AlarmActive : BOOL;
		AlarmActiveColour : USINT;
	END_STRUCT;
	UDT_InclinoSensor_ALM : 	STRUCT
		dummy : USINT;
	END_STRUCT;
	UDT_InclinoSensor_IO : 	STRUCT
		DataMSB : USINT;
		DataLSB : USINT;
		SetCenterPoint : USINT;
	END_STRUCT;
END_TYPE
```

#### UDT_FieldMotor.typ
```iecst
TYPE
	UDT_FieldMotor_CS : 	STRUCT
		Home : BOOL;
		MoveAbsolute : BOOL;
		MoveJogNeg : BOOL;
		MoveJogPos : BOOL;
		Power : BOOL;
		Stop : BOOL;
		StopGame : BOOL;
		ErrorAcknowledge : BOOL;
		Start : BOOL;
		Interlock : BOOL;
		Initialize : BOOL;
		SetCenterPoint : BOOL;
	END_STRUCT;
	UDT_FieldMotor_HMI : 	STRUCT
		MoveAbsolute : BOOL;
		MoveJogNeg : BOOL;
		MoveJogPos : BOOL;
		Power : BOOL;
		IncreaseJogSpeed : BOOL;
		DecreaseJogSpeed : BOOL;
		ErrorAcknowledge : BOOL;
	END_STRUCT;
	UDT_FieldMotor_PAR : 	STRUCT
		Acceleration : REAL;
		Deceleration : REAL;
		JogVelocity : REAL;
		Velocity : REAL;
		Position : REAL;
	END_STRUCT;
	UDT_FieldMotor_STS : 	STRUCT
		Disabled : BOOL;
		Idle : BOOL;
		Initializing : BOOL;
		Running : BOOL;
		Moving : BOOL;
		StandStill : BOOL;
		AtTargetPosition : BOOL;
		AutoActive : BOOL;
		StateInt : USINT;
		AlarmActive : BOOL;
		ActPosition : REAL;
		ActVelocity : REAL;
		Interlocked : BOOL;
		PowerOn : BOOL;
		EndButtonHit : BOOL;
		TimerStarted : BOOL;
		TimerEnded : BOOL;
		ReferencePosition : REAL;
		AlarmActiveColour : USINT;
	END_STRUCT;
	UDT_FieldMotor_ALM : 	STRUCT
		MotorError : BOOL;
		ErrorID : UINT;
		ErrorText : ARRAY[0..3]OF STRING[79];
	END_STRUCT;
	UDT_FieldMotor_IO : 	STRUCT
		EndButton : BOOL;
		Power : BOOL;
		Home : BOOL;
		ErrorAcknowledge : BOOL;
		MoveJogNeg : BOOL;
		MoveJogPos : BOOL;
		Stop : BOOL;
		MoveAbsolute : BOOL;
		Acceleration : REAL;
		Deceleration : REAL;
		JogVelocity : REAL;
		Velocity : REAL;
		Position : REAL;
	END_STRUCT;
END_TYPE
```

#### UDT_Shooter.typ
```iecst
TYPE
	UDT_Shooter_CS : 	STRUCT
		Interlock : BOOL;
		EnableFan : BOOL;
		Shoot : BOOL;
		StopGame : BOOL;
		Start : BOOL;
		AutoMode : BOOL;
	END_STRUCT;
	UDT_Shooter_HMI : 	STRUCT
		EnableFan : BOOL;
		Shoot : BOOL;
		IncreaseIntensity : BOOL;
		DecreaseIntensity : BOOL;
	END_STRUCT;
	UDT_Shooter_PAR : 	STRUCT
		Intensity : REAL;
	END_STRUCT;
	UDT_Shooter_STS : 	STRUCT
		Disabled : BOOL;
		Idle : BOOL;
		Interlocked : BOOL;
		AlarmActive : BOOL;
		AutoActive : BOOL;
		Shooting : BOOL;
		StateInt : USINT;
		AlarmActiveColour : USINT;
	END_STRUCT;
	UDT_Shooter_ALM : 	STRUCT
		dummy : BOOL;
	END_STRUCT;
	UDT_Shooter_IO : 	STRUCT
		EnableFan : BOOL;
		Shoot : BOOL;
	END_STRUCT;
END_TYPE
```

#### FB_PaddleMotor.c
```c
/*********************************************************************************
 * Copyright: MyAutomation-IT
 * Author:    raivo
 * Created:   April 22, 2026/5:57 PM
 *********************************************************************************/
#include <bur/plctypes.h>
#include <standard.h>
#include "CommonTypes.h"

#ifdef __cplusplus
	extern "C"
	{
#endif
	#include "Library.h"
#ifdef __cplusplus
	};
#endif

#define ENDBUTTON_BITMASK 0x2
#define MIDDLE_POSITION 1450

/* dynamic braking offset (speed-dependent approach distance) */
#define STOPPING_OFFSET ((PaddleMotor->STS.ActVelocity * PaddleMotor->STS.ActVelocity) / 46000)

/* mechanical reference correction */
#define REFERENCE_OFFSET 25

#define PaddleMotor inst->PaddleMotor

_LOCAL TON_typ PaddleMotorTimer;

void FB_PaddleMotor(struct FB_PaddleMotor* inst)
{
	/* input decode */
	PaddleMotor->IO.EndButton = !((inst->digitalInput & ENDBUTTON_BITMASK) >> 1);

	/* stop request handling */
	if(PaddleMotor->CS.StopGame && !PaddleMotor->STS.AlarmActive && !PaddleMotor->STS.Interlocked)
	{
		PaddleMotor->STS.StateInt = STATE_STOPPING;
	}

	PaddleMotor->STS.AlarmActiveColour = PaddleMotor->STS.AlarmActive ? RED_COLOUR : GREEN_COLOUR;

	switch(PaddleMotor->STS.StateInt)
	{
		case STATE_DISABLED:
			/* full reset of outputs and internal flags */
			PaddleMotor->STS.Disabled = 1;

			PaddleMotor->CS.Power = 0;
			PaddleMotor->CS.Home = 0;
			PaddleMotor->CS.MoveJogNeg = 0;
			PaddleMotor->CS.MoveJogPos = 0;
			PaddleMotor->CS.MoveAbsolute = 0;

			PaddleMotor->HMI.MoveJogNeg = 0;
			PaddleMotor->HMI.MoveJogPos = 0;

			PaddleMotor->STS.TimerStarted = 0;
			PaddleMotor->STS.TimerEnded = 0;
			PaddleMotor->STS.ReferencePosition = 0;
			PaddleMotor->STS.ReferenceSet = 0;
			PaddleMotor->STS.EndButtonHit = 0;

			/* reset homing timer */
			PaddleMotorTimer.IN = 0;
			TON(&PaddleMotorTimer);

			if(PaddleMotor->CS.Initialize && !PaddleMotor->STS.AlarmActive && !PaddleMotor->STS.Interlocked)
			{
				PaddleMotor->STS.StateInt = STATE_INITIALIZING;
			}
			break;
		case STATE_INITIALIZING:
			/* enable drive + default parameters */
			PaddleMotor->STS.Initializing = 1;
			PaddleMotor->STS.Disabled = 0;
			PaddleMotor->PAR.Acceleration = MAX_ACC_DEC;
			PaddleMotor->PAR.Deceleration = MAX_ACC_DEC;
			PaddleMotor->PAR.JogVelocity = STD_VELOCITY;
			PaddleMotor->PAR.Velocity = STD_VELOCITY;

			PaddleMotor->CS.Power = 1;
			PaddleMotor->CS.Stop = 0;

			/* disable manual commands during init */
			PaddleMotor->HMI.MoveJogNeg = 0;
			PaddleMotor->HMI.MoveJogPos = 0;

			/* homing start condition */
			if(!PaddleMotor->IO.EndButton && !PaddleMotor->STS.EndButtonHit)
			{
				PaddleMotor->CS.Home = 1;
				if(!PaddleMotor->STS.TimerStarted)
				{
					PaddleMotorTimer.IN = 1;
					PaddleMotor->STS.TimerStarted = 1;
				}
				PaddleMotorTimer.PT = MS_100;
				TON(&PaddleMotorTimer);

				if(PaddleMotorTimer.Q)
				{
					PaddleMotor->CS.Home = 0;
					PaddleMotor->CS.MoveJogPos = 1;
				}
			}
			/* end switch reached */
			else if(PaddleMotor->IO.EndButton && !PaddleMotor->STS.EndButtonHit)
			{
				PaddleMotorTimer.IN = 0;
				PaddleMotor->STS.TimerStarted = 0;

				PaddleMotor->CS.MoveJogPos = 0;
				PaddleMotor->STS.EndButtonHit = 1;
				PaddleMotor->CS.Home = 1;

				PaddleMotorTimer.IN = 1;
				PaddleMotor->STS.TimerStarted = 1;
			}
			/* post homing alignment */
			else if(PaddleMotor->STS.EndButtonHit)
			{
				if(PaddleMotorTimer.Q && !PaddleMotor->STS.TimerEnded)
				{
					PaddleMotor->STS.TimerEnded = 1;

				}
				/* set reference position */
				if(PaddleMotor->STS.TimerEnded && !PaddleMotor->STS.ReferenceSet)
				{
					PaddleMotor->STS.ReferenceSet = 1;
					PaddleMotor->CS.Home = 0;

					PaddleMotor->STS.ReferencePosition = PaddleMotor->STS.ActPosition + REFERENCE_OFFSET;
					PaddleMotor->PAR.Position = PaddleMotor->STS.ReferencePosition - MIDDLE_POSITION;
					PaddleMotor->CS.MoveAbsolute = 1;
				}
				/* finish init when position reached */
				if(PaddleMotor->STS.ActPosition <= PaddleMotor->PAR.Position && !PaddleMotor->STS.AlarmActive && !PaddleMotor->STS.Interlocked)
				{
					PaddleMotor->CS.MoveAbsolute = 0;
					PaddleMotor->STS.StateInt = STATE_IDLE;
				}
			}
			break;
		case STATE_IDLE:
			/* idle state reset */
			PaddleMotor->STS.Initializing = 0;
			PaddleMotor->STS.Idle = 1;

			PaddleMotor->CS.MoveAbsolute = 0;
			PaddleMotor->CS.MoveJogNeg = 0;
			PaddleMotor->CS.MoveJogPos = 0;
			PaddleMotor->HMI.MoveJogPos = 0;
			PaddleMotor->HMI.MoveAbsolute = 0;
			PaddleMotor->HMI.MoveJogNeg = 0;

			if(PaddleMotor->CS.Start && !PaddleMotor->STS.AlarmActive && !PaddleMotor->STS.Interlocked)
			{
				PaddleMotor->STS.StateInt = STATE_RUNNING;
			}
			break;
		case STATE_RUNNING:
			/* active motion state */
			PaddleMotor->STS.Running = 1;
			PaddleMotor->STS.Idle = 0;

			if(!PaddleMotor->STS.AutoActive)
			{
				/* manual control mode */
				PaddleMotor->CS.MoveAbsolute = 0;
				PaddleMotor->CS.MoveJogNeg = 0;
				PaddleMotor->CS.MoveJogPos = 0;

				/* jog speed tuning */
				if(PaddleMotor->HMI.IncreaseJogSpeed && PaddleMotor->PAR.JogVelocity < MAX_VELOCITY)
				{
					PaddleMotor->PAR.JogVelocity++;
				}
				else if(PaddleMotor->HMI.DecreaseJogSpeed && PaddleMotor->PAR.JogVelocity > MIN_VELOCITY)
				{
					PaddleMotor->PAR.JogVelocity--;
				}
			}
			else
			{
				/* auto mode overrides HMI input */
				PaddleMotor->HMI.MoveAbsolute = 0;
				PaddleMotor->HMI.MoveJogNeg = 0;
				PaddleMotor->HMI.MoveJogPos = 0;
			}

			/* lower limit protection */
			if(PaddleMotor->STS.ActPosition < MIN_POSITION + STOPPING_OFFSET)
			{
				PaddleMotor->CS.MoveJogNeg = 0;
				PaddleMotor->HMI.MoveJogNeg = 0;
				PaddleMotor->PAR.Position = PaddleMotor->STS.ActPosition + 100;
			}
			/* upper limit protection */
			else if(PaddleMotor->IO.EndButton || PaddleMotor->STS.ActPosition >= (PaddleMotor->STS.ReferencePosition - (STOPPING_OFFSET + 100)))
			{
				PaddleMotor->CS.MoveJogPos = 0;
				PaddleMotor->HMI.MoveJogPos = 0;
				PaddleMotor->PAR.Position = PaddleMotor->STS.ReferencePosition - 100;
			}
			break;
		case STATE_STOPPING:
			/* safe stop state */
			PaddleMotor->STS.Running = 0;
			PaddleMotor->STS.Initializing = 0;
			PaddleMotor->STS.Idle = 0;

			PaddleMotor->CS.MoveAbsolute = 0;
			PaddleMotor->CS.MoveJogNeg = 0;
			PaddleMotor->CS.MoveJogPos = 0;
			PaddleMotor->CS.Stop = 1;

			PaddleMotor->HMI.MoveJogNeg = 0;
			PaddleMotor->HMI.MoveJogPos = 0;

			if(PaddleMotor->STS.StandStill && !PaddleMotor->STS.Interlocked)
			{
				PaddleMotor->STS.StateInt = STATE_DISABLED;
			}
			break;
	}

	/* IO mapping */
	PaddleMotor->IO.Power = PaddleMotor->CS.Power;
	PaddleMotor->IO.Home = PaddleMotor->CS.Home;

	PaddleMotor->IO.JogVelocity = PaddleMotor->PAR.JogVelocity;
	PaddleMotor->IO.Acceleration = PaddleMotor->PAR.Acceleration;
	PaddleMotor->IO.Deceleration = PaddleMotor->PAR.Deceleration;
	PaddleMotor->IO.Velocity = PaddleMotor->PAR.Velocity;
	PaddleMotor->IO.Position = PaddleMotor->PAR.Position;

	PaddleMotor->IO.ErrorAcknowledge = PaddleMotor->HMI.ErrorAcknowledge ^ PaddleMotor->CS.ErrorAcknowledge;
	PaddleMotor->IO.MoveJogPos = PaddleMotor->CS.MoveJogPos ^ PaddleMotor->HMI.MoveJogPos;
	PaddleMotor->IO.MoveJogNeg = PaddleMotor->CS.MoveJogNeg ^ PaddleMotor->HMI.MoveJogNeg;
	PaddleMotor->IO.MoveAbsolute = PaddleMotor->CS.MoveAbsolute ^ PaddleMotor->HMI.MoveAbsolute;

	/* alarm source */
	PaddleMotor->STS.AlarmActive = PaddleMotor->ALM.MotorError;

	/* derived motion states */
	PaddleMotor->STS.StandStill = (int)PaddleMotor->STS.ActVelocity == 0;
	PaddleMotor->STS.Moving = !PaddleMotor->STS.StandStill;

	PaddleMotor->STS.AutoActive = PaddleMotor->CS.AutoMode;

}
```

#### FB_DistanceSensor.c
```c
/*********************************************************************************
 * Copyright: MyAutomation-IT
 * Author:    raivo
 * Created:   April 22, 2026/5:57 PM
 *********************************************************************************/
#include <bur/plctypes.h>
#include "CommonTypes.h"
#ifdef __cplusplus
	extern "C"
	{
#endif
	#include "Library.h"
#ifdef __cplusplus
	};
#endif

void FB_DistanceSensor(struct FB_DistanceSensor* inst)
{
	/* sensor list abstraction */
	UDT_DistanceSensor* sensors[NUM_SENSORS] =
	{
		inst->DistanceSensorLeft,
		inst->DistanceSensorMiddle,
		inst->DistanceSensorRight
	};

	int i;
	for(i = 0; i < NUM_SENSORS; i++)
	{
		/* combine MSB/LSB */
		INT Distance = ((sensors[i]->IO.DataMSB << SHIFT_BYTE) | sensors[i]->IO.DataLSB);

		/* clamp invalid sensor range */
		if(Distance > BALL_MAX_DISTANCE && Distance < OVERLOAD)
		{
			sensors[i]->STS.TooFar = 1;
			sensors[i]->STS.TooClose = 0;
			sensors[i]->ALM.OutOfBounds = 1;
		}
		else if(Distance < BALL_MIN_DISTANCE && Distance > UNDERLOAD)
		{
			sensors[i]->STS.TooClose = 1;
			sensors[i]->STS.TooFar = 0;
			sensors[i]->ALM.OutOfBounds = 1;
		}
		else if(Distance <= UNDERLOAD || Distance >= OVERLOAD)
		{
			sensors[i]->STS.Distance = 0;
			sensors[i]->ALM.OutOfBounds = 0;
			sensors[i]->STS.TooClose = 0;
			sensors[i]->STS.TooFar = 0;
		}
		else
		{
			sensors[i]->STS.TooClose = 0;
			sensors[i]->STS.TooFar = 0;
			sensors[i]->ALM.OutOfBounds = 0;
			sensors[i]->STS.Distance = Distance;
		}

		/* decode sensor IO bits */
		sensors[i]->IO.OUT1 = sensors[i]->IO.SensorInfo & OUT1_BITMASK;
		sensors[i]->IO.OUT2 = (sensors[i]->IO.SensorInfo & OUT2_BITMASK) >> 1;
		sensors[i]->STS.BallDetected = sensors[i]->STS.Distance >= BALL_MIN_DISTANCE && sensors[i]->STS.Distance <= BALL_MAX_DISTANCE;
		sensors[i]->STS.DeviceStatus = (sensors[i]->IO.SensorInfo & DEVICE_STATUS_BITMASK) >> 4;

		/* alarm indication */
		sensors[i]->STS.AlarmActiveColour = sensors[i]->STS.AlarmActive ? RED_COLOUR : GREEN_COLOUR;

		if(sensors[i]->STS.DeviceStatus == SENSOR_FAILURE || sensors[i]->ALM.OutOfBounds)
		{
			sensors[i]->STS.AlarmActive = 1;
		}
		else if(sensors[i]->STS.DeviceStatus != SENSOR_FAILURE)
		{
			sensors[i]->STS.AlarmActive = 0;
		}
	}

}
```

#### FB_Shooter.c
```c
/*********************************************************************************
 * Copyright: MyAutomation-IT
 * Author:    raivo
 * Created:   April 22, 2026/5:57 PM
 *********************************************************************************/
#include <bur/plctypes.h>
#include "CommonTypes.h"
#ifdef __cplusplus
	extern "C"
	{
#endif
	#include "Library.h"
#ifdef __cplusplus
	};
#endif

#define STATE_SHOOTING 50

#define Shooter inst->Shooter

/* TODO: Add your comment here */
void FB_Shooter(struct FB_Shooter* inst)
{
	if(Shooter->CS.StopGame && !Shooter->STS.Interlocked)
	{
		Shooter->STS.StateInt = STATE_DISABLED;
	}

	Shooter->STS.AlarmActiveColour = GREEN_COLOUR;
	if(Shooter->STS.AlarmActive)
	{
		Shooter->STS.AlarmActiveColour = RED_COLOUR;
	}

	switch (Shooter->STS.StateInt)
	{
		case STATE_DISABLED:
			Shooter->STS.Disabled = 1;
			Shooter->STS.Idle = 0;

			Shooter->HMI.Shoot = 0;
			Shooter->HMI.EnableFan = 0;

			Shooter->CS.Shoot = 0;
			Shooter->CS.EnableFan = 0;
			Shooter->CS.Interlock = 0;

			if(Shooter->HMI.IncreaseIntensity)
			{
				Shooter->PAR.Intensity += 0.1;
			}
			else if(Shooter->HMI.DecreaseIntensity)
			{
				Shooter->PAR.Intensity -= 0.1;
			}
			if(Shooter->CS.Start && !Shooter->STS.AlarmActive && !Shooter->STS.Interlocked)
			{
				Shooter->STS.StateInt = STATE_IDLE;
			}
			break;
		case STATE_IDLE:
			Shooter->STS.Idle = 1;
			Shooter->STS.Disabled = 0;
			Shooter->STS.Shooting = 0;

			Shooter->CS.Interlock = 0;

			if(Shooter->STS.AutoActive)
			{
				Shooter->HMI.Shoot = 0;
			}
			else
			{
				if(!Shooter->HMI.EnableFan)
				{
					Shooter->CS.Interlock = 1;
				}
				Shooter->CS.Shoot = 0;
			}

			if((Shooter->HMI.Shoot ^ Shooter->CS.Shoot) == 1 && !Shooter->STS.AlarmActive && !Shooter->STS.Interlocked)
			{
				Shooter->STS.StateInt = STATE_SHOOTING;
			}
			break;
		case STATE_SHOOTING:
			Shooter->STS.Shooting = 1;

			if(!Shooter->CS.Shoot && !Shooter->HMI.Shoot && !Shooter->STS.AlarmActive && !Shooter->STS.Interlocked)
			{
				Shooter->STS.StateInt = STATE_IDLE;
			}
			break;
	}

	if(!Shooter->STS.Interlocked && !Shooter->STS.AlarmActive)
	{
		Shooter->IO.Shoot = Shooter->HMI.Shoot ^ Shooter->CS.Shoot;
	}

	Shooter->IO.EnableFan = Shooter->HMI.EnableFan ^ Shooter->CS.EnableFan;

	Shooter->STS.Interlocked = Shooter->CS.Interlock;
	Shooter->STS.AutoActive = Shooter->CS.AutoMode;

	inst->digitalOutput = 0;
	inst->digitalOutput |= (Shooter->IO.Shoot << 3);
	inst->digitalOutput |= Shooter->IO.EnableFan;

}
```

#### FB_FieldMotor.c
```c
/*********************************************************************************
 * Copyright: MyAutomation-IT
 * Author:    raivo
 * Created:   April 22, 2026/5:57 PM
 *********************************************************************************/
#include <bur/plctypes.h>
#include <standard.h>
#include "CommonTypes.h"
#ifdef __cplusplus
	extern "C"
	{
#endif
	#include "Library.h"
#ifdef __cplusplus
	};
#endif

#define ENDBUTTON_BITMASK 0x4
#define MIN_POSITION FieldMotor->STS.ReferencePosition - 2800

#define FieldMotor inst->FieldMotor

_LOCAL TON_typ FieldMotorTimer;

/* TODO: Add your comment here */
void FB_FieldMotor(struct FB_FieldMotor* inst)
{
	//FieldMotorTimer.IN = 0;
	if(FieldMotor->STS.AlarmActive)
	{
		FieldMotor->STS.AlarmActiveColour = RED_COLOUR;
		//FieldMotor->CS.Stop = 1;
	}
	FieldMotor->IO.EndButton = !((inst->digitalInput & ENDBUTTON_BITMASK) >> 2);

	if(FieldMotor->CS.StopGame)
	{
		FieldMotor->STS.StateInt = STATE_STOPPING;
	}

	FieldMotor->STS.AlarmActiveColour = GREEN_COLOUR;

	switch(FieldMotor->STS.StateInt)
	{
		case STATE_DISABLED:
			FieldMotor->CS.Power = 0;
			FieldMotor->CS.Home = 0;
			FieldMotor->CS.MoveJogNeg = 0;
			FieldMotor->CS.MoveJogPos = 0;
			FieldMotor->CS.MoveAbsolute = 0;

			FieldMotor->STS.Disabled = 1;
			FieldMotor->STS.EndButtonHit = 0;
			FieldMotor->STS.TimerStarted = 0;
			FieldMotor->STS.TimerEnded = 0;
			FieldMotor->STS.ReferencePosition = 0;
			FieldMotor->STS.AtTargetPosition = 0;

			if(FieldMotor->CS.Initialize && !FieldMotor->STS.AlarmActive && !FieldMotor->STS.Interlocked)
			{
				FieldMotor->STS.StateInt = STATE_INITIALIZING;
			}
			break;
		case STATE_INITIALIZING:
			FieldMotor->CS.Power = 1;
			FieldMotor->CS.Stop = 0;

			FieldMotor->STS.Initializing = 1;
			FieldMotor->STS.Disabled = 0;

			FieldMotor->PAR.Acceleration = MAX_ACC_DEC;
			FieldMotor->PAR.Deceleration = MAX_ACC_DEC;
			FieldMotor->PAR.JogVelocity = STD_VELOCITY;
			FieldMotor->PAR.Velocity = STD_VELOCITY;

			FieldMotorTimer.PT = MS_100;
			TON(&FieldMotorTimer);

			if(!FieldMotor->IO.EndButton && !FieldMotor->STS.EndButtonHit)
			{
				if(!FieldMotor->STS.TimerStarted)
				{
					FieldMotorTimer.IN = 1;
					FieldMotor->STS.TimerStarted = 1;
					FieldMotor->CS.Home = 1;
				}
				if(FieldMotorTimer.Q)
				{
					FieldMotorTimer.IN = 0;
					FieldMotor->CS.Home = 0;
					FieldMotor->CS.MoveJogPos = 1;
				}
			}
			else if(FieldMotor->IO.EndButton && !FieldMotor->STS.EndButtonHit)
			{
				FieldMotor->CS.MoveJogPos = 0;
				FieldMotor->STS.EndButtonHit = 1;
				FieldMotor->CS.Home = 1;
				FieldMotor->CS.SetCenterPoint = 1;

				FieldMotorTimer.IN = 1;
			}
			else if(FieldMotor->STS.EndButtonHit)
			{
				if(FieldMotorTimer.Q)
				{
					FieldMotorTimer.IN = 0;
					FieldMotor->STS.TimerStarted = 0;
					FieldMotor->CS.Home = 0;
					FieldMotor->CS.SetCenterPoint = 0;
					FieldMotor->CS.MoveJogNeg = 1;
				}
				if(FieldMotor->STS.AtTargetPosition && !FieldMotor->STS.AlarmActive && !FieldMotor->STS.Interlocked)
				{
					FieldMotor->CS.MoveJogNeg = 0;
					FieldMotor->STS.StateInt = STATE_IDLE;
				}

			}
			break;
		case STATE_IDLE:
			FieldMotor->STS.Initializing = 0;
			FieldMotor->STS.Idle = 1;

			FieldMotor->CS.MoveAbsolute = 0;
			FieldMotor->CS.MoveJogNeg = 0;
			FieldMotor->CS.MoveJogPos = 0;
			FieldMotor->CS.Power = 0;

			if(FieldMotor->CS.Start && !FieldMotor->STS.AlarmActive && !FieldMotor->STS.Interlocked)
			{
				FieldMotor->STS.StateInt = STATE_RUNNING;
			}
			break;
		case STATE_RUNNING:
			FieldMotor->STS.Running = 1;
			FieldMotor->STS.Idle = 0;
			FieldMotor->CS.Power = 1;

			if(!FieldMotor->STS.AutoActive)
			{
				FieldMotor->CS.MoveAbsolute = 0;
				FieldMotor->CS.MoveJogNeg = 0;
				FieldMotor->CS.MoveJogPos = 0;
				//control parameters
				if(FieldMotor->HMI.IncreaseJogSpeed && FieldMotor->PAR.JogVelocity < MAX_VELOCITY)
				{
					FieldMotor->PAR.JogVelocity++;
				}
				else if(FieldMotor->HMI.DecreaseJogSpeed && FieldMotor->PAR.JogVelocity > 0)
				{
					FieldMotor->PAR.JogVelocity--;
				}
			}
			else
			{
				FieldMotor->HMI.MoveAbsolute = 0;
				FieldMotor->HMI.MoveJogNeg = 0;
				FieldMotor->HMI.MoveJogPos = 0;
			}
			if(FieldMotor->IO.EndButton)
			{
				FieldMotor->CS.MoveJogPos = 0;
				FieldMotor->HMI.MoveJogPos = 0;
				FieldMotor->CS.MoveAbsolute = 0;
			}
			break;
		case STATE_STOPPING:
			FieldMotor->STS.Running = 0;
			FieldMotor->STS.Idle = 0;
			FieldMotor->STS.Initializing = 0;

			FieldMotor->CS.MoveAbsolute = 0;
			FieldMotor->CS.MoveJogNeg = 0;
			FieldMotor->CS.MoveJogPos = 0;
			FieldMotor->CS.Stop = 1;

			if(FieldMotor->STS.StandStill && !FieldMotor->STS.Interlocked)
			{
				FieldMotor->STS.StateInt = STATE_DISABLED;
			}
			break;
	}

	//io mapping

	FieldMotor->IO.Power = FieldMotor->CS.Power;
	FieldMotor->IO.Home = FieldMotor->CS.Home;
	FieldMotor->IO.Stop = FieldMotor->CS.Stop;

	FieldMotor->IO.JogVelocity = FieldMotor->PAR.JogVelocity;
	FieldMotor->IO.Acceleration = FieldMotor->PAR.Acceleration;
	FieldMotor->IO.Deceleration = FieldMotor->PAR.Deceleration;
	FieldMotor->IO.Velocity = FieldMotor->PAR.Velocity;
	FieldMotor->IO.Position = FieldMotor->PAR.Position;
	FieldMotor->IO.ErrorAcknowledge = FieldMotor->HMI.ErrorAcknowledge;
	FieldMotor->IO.MoveJogPos = FieldMotor->CS.MoveJogPos ^ FieldMotor->HMI.MoveJogPos;
	FieldMotor->IO.MoveJogNeg = FieldMotor->CS.MoveJogNeg ^ FieldMotor->HMI.MoveJogNeg;
	FieldMotor->IO.MoveAbsolute = FieldMotor->CS.MoveAbsolute ^ FieldMotor->HMI.MoveAbsolute;

	FieldMotor->STS.AlarmActive = FieldMotor->ALM.MotorError;
	FieldMotor->STS.StandStill = (int)FieldMotor->STS.ActVelocity == 0;
	FieldMotor->STS.Moving = !FieldMotor->STS.StandStill;

}
```

#### FB_InclinoSensor.c
```c
/*********************************************************************************
 * Copyright: MyAutomation-IT
 * Author:    raivo
 * Created:   April 22, 2026/5:57 PM
 *********************************************************************************/
#include <bur/plctypes.h>
#include <standard.h>
#include "CommonTypes.h"
#ifdef __cplusplus
	extern "C"
	{
#endif
	#include "Library.h"
#ifdef __cplusplus
	};
#endif

#define TO_DEGREES 100
#define SHIFT_BYTE 8

#define InclinoSensor inst->InclinoSensor

void FB_InclinoSensor(struct FB_InclinoSensor* inst)
{
	//Combining MSB and LSB with bitwise operators to show the value. Dividing by 100 to convert to degrees and explicit casting to float to show CurrentAngle as accurate as possible.
	InclinoSensor->STS.CurrentAngle = (float)((INT)((InclinoSensor->IO.DataMSB << SHIFT_BYTE) | InclinoSensor->IO.DataLSB)) / TO_DEGREES;

	InclinoSensor->STS.AlarmActiveColour = GREEN_COLOUR;
	if(InclinoSensor->STS.AlarmActive)
	{
		InclinoSensor->STS.AlarmActiveColour = RED_COLOUR;
	}
	InclinoSensor->IO.SetCenterPoint = 7;
	if(InclinoSensor->CS.SetCenterPoint)
	{

		InclinoSensor->IO.SetCenterPoint = 3;
	}
}
```

#### FB_BallControl.c
```c
/*********************************************************************************
 * Copyright: MyAutomation-IT
 * Author:    raivo
 * Created:   April 22, 2026/5:57 PM
 *********************************************************************************/
#include <bur/plctypes.h>
#include <standard.h>
#include "CommonTypes.h"
#ifdef __cplusplus
	extern "C"
	{
#endif
	#include "Library.h"
#ifdef __cplusplus
	};
#endif

#define BallControl inst->BallControl
#define PaddleMotor inst->PaddleMotor
#define Shooter inst->Shooter
#define DistanceSensorLeft inst->DistanceSensorLeft
#define DistanceSensorMiddle inst->DistanceSensorMiddle
#define DistanceSensorRight inst->DistanceSensorRight

_LOCAL TON_typ SpeedTimer;
_LOCAL TON_typ ShootTimer;
_LOCAL TON_typ ShootDelayTimer;
_LOCAL TON_typ NewShootCycleTimer;

void FB_BallControl(struct FB_BallControl* inst)
{
	/* reset per cycle */
	BallControl->STS.ShootCycleCompleted = 0;

	if(BallControl->CS.StopGame && !BallControl->STS.Interlocked)
	{
		/* immediate stop override */
		BallControl->STS.StateInt = STATE_STOPPING;
		Shooter->PAR.Intensity = 3;
	}

	switch(BallControl->STS.StateInt)
	{
		case STATE_DISABLED:
		{
			BallControl->CS.Shoot = 0;

			/* Allow parameter tuning only when inactive */
			if(Shooter->HMI.IncreaseIntensity && Shooter->PAR.Intensity < MAX_INTENSITY)
			{
				Shooter->PAR.Intensity += 0.002;
			}
			else if(Shooter->HMI.DecreaseIntensity && Shooter->PAR.Intensity > MIN_INTENSITY)
			{
				Shooter->PAR.Intensity -= 0.002;
			}

			if(BallControl->STS.Initializing)
			{
				BallControl->STS.StateInt = STATE_INITIALIZING;
			}
			break;
		}
		case STATE_INITIALIZING:
		{
			BallControl->STS.PrevShootState = 0;
			BallControl->STS.ShootState = 0;
			BallControl->STS.GameOver = 0;
			BallControl->STS.FirstRun = 1;
			if(BallControl->STS.Idle)
			{
				BallControl->STS.StateInt = STATE_IDLE;
			}
			break;
		}
		case STATE_IDLE:
		{
			NewShootCycleTimer.IN = 0;
			if(BallControl->STS.Running)
			{
				BallControl->STS.StateInt = STATE_RUNNING;
			}
			break;
		}
		case STATE_RUNNING:
		{
			if(BallControl->STS.AutoActive)
			{
				/* auto mode outputs */
				PaddleMotor->CS.MoveAbsolute = 0;
				Shooter->CS.EnableFan = 1;
				PaddleMotor->PAR.Velocity = AUTOMODE_VELOCITY;

				/* shoot delay release */
				if(ShootDelayTimer.Q)
				{
					BallControl->CS.Shoot = 0;
					ShootDelayTimer.IN = 0;
				}

				BallControl->STS.NewShootCycleTimerET = NewShootCycleTimer.ET;
				switch(BallControl->STS.ShootState)
				{
					case 0:
					{
						SpeedTimer.IN = 0;

						if(BallControl->STS.FirstRun)
						{
							if(DistanceSensorRight->STS.BallDetected)
							{
								BallControl->PAR.DesiredPosition = MIN_POSITION + ((DistanceSensorRight->STS.Distance - MIN_FIELD_DISTANCE) * MM_TO_POSITION);

								BallControl->STS.ShootState = 5;
								BallControl->STS.FirstRun = 0;
							}
						}
						else
						{
							/* cycle timeout -> game over */
							if(NewShootCycleTimer.Q)
							{
								NewShootCycleTimer.IN = 0;
								BallControl->STS.GameOver = 1;
							}
							else if(NewShootCycleTimer.ET >= MS_500)
							{
								if(DistanceSensorRight->STS.BallDetected)
								{
									BallControl->PAR.DesiredPosition = MIN_POSITION + ((DistanceSensorRight->STS.Distance - MIN_FIELD_DISTANCE) * MM_TO_POSITION);

									NewShootCycleTimer.IN = 0;
									BallControl->STS.ShootState = 5;
								}
							}

						}
					}
					break;

					case 5:
						/* speed measurement start */
						SpeedTimer.PT = MS_1000;
						SpeedTimer.IN = 1;
						BallControl->STS.ShootState = 10;
					break;

					case 10:
						if(DistanceSensorMiddle->STS.BallDetected)
						{
							BallControl->PAR.DesiredPosition = MIN_POSITION + ((DistanceSensorMiddle->STS.Distance - MIN_FIELD_DISTANCE) * MM_TO_POSITION);

							/* range validation */
							if(BallControl->PAR.DesiredPosition >= MIN_POSITION && BallControl->PAR.DesiredPosition <= MAX_POSITION)
								{
									//reserved motion trigger:
									//PaddleMotor->PAR.Position = BallControl->PAR.DesiredPosition;
									//PaddleMotor->CS.MoveAbsolute = 1;
								}
							BallControl->STS.ShootState = 20;
						}
						break;

					case 20:
						if(DistanceSensorLeft->STS.BallDetected)
						{
							/* velocity calculation window */
							SpeedTimer.IN = 0;

							if(SpeedTimer.ET > 0)
							{
								BallControl->STS.BallVelocity = (DISTANCE_BETWEEN_SENSORS_MM * 2.0f) / (float)SpeedTimer.ET; // m/s
								BallControl->STS.TimeToPaddleMS = SpeedTimer.ET;

								ShootTimer.PT = BallControl->STS.TimeToPaddleMS;
							}
							else
							{
								BallControl->STS.BallVelocity = 0.0f;
								ShootTimer.PT = 0;
							}

							ShootTimer.IN = 1;

							BallControl->PAR.DesiredPosition = MIN_POSITION + ((DistanceSensorLeft->STS.Distance - MIN_FIELD_DISTANCE) * MM_TO_POSITION);

							if(BallControl->PAR.DesiredPosition >= MIN_POSITION && BallControl->PAR.DesiredPosition <= MAX_POSITION)
							{
								// reserved motion trigger:
								//PaddleMotor->PAR.Position = BallControl->PAR.DesiredPosition;
								//PaddleMotor->CS.MoveAbsolute = 1;
							}

							BallControl->STS.ShootState = 30;
						}
					break;

					case 30:
						if(ShootTimer.Q)
						{
							/* fire command pulse */
							BallControl->CS.Shoot = 1;

							ShootTimer.IN = 0;

							BallControl->STS.ShootState = 0;
							ShootDelayTimer.PT = (DINT)(MS_50 * Shooter->PAR.Intensity);

							ShootDelayTimer.IN = 1;
						}
					break;
				}

				/* cycle completion detection */
				if (BallControl->STS.PrevShootState == 30 && BallControl->STS.ShootState == 0)
				{
					NewShootCycleTimer.IN = 1;
					NewShootCycleTimer.PT = GAME_OVER_TRIGGER_MS;
					BallControl->STS.ShootCycleCompleted = 1;
				}

				TON(&ShootTimer);
				TON(&SpeedTimer);
				TON(&ShootDelayTimer);
				TON(&NewShootCycleTimer);
			}
			else
			{
				BallControl->CS.Shoot = 0;
			}
			break;
		}
		case STATE_STOPPING:
		{
			if(BallControl->STS.Disabled)
			{
				BallControl->STS.StateInt = STATE_DISABLED;
			}
			break;
		}
	}

	/* latch previous shoot state */
	BallControl->STS.PrevShootState = BallControl->STS.ShootState;

	BallControl->STS.PaddlePositionMM = (INT)((MAX_PADDLE_DISTANCE_TICKS - (PaddleMotor->STS.ReferencePosition - PaddleMotor->STS.ActPosition)) * TICKS_TO_MM);

	/* command forwarding */
	PaddleMotor->CS.Initialize = BallControl->CS.Initialize;
	PaddleMotor->CS.Start = BallControl->CS.Start;
	PaddleMotor->CS.StopGame = BallControl->CS.StopGame;
	PaddleMotor->CS.AutoMode = BallControl->CS.AutoMode;
	PaddleMotor->CS.ErrorAcknowledge = BallControl->CS.ErrorAcknowledge;

	Shooter->CS.Start = BallControl->CS.Start;
	Shooter->CS.StopGame = BallControl->CS.StopGame;
	Shooter->CS.AutoMode = BallControl->CS.AutoMode;
	Shooter->CS.Shoot = BallControl->CS.Shoot;

	/* subsystem state mapping */
	BallControl->STS.Idle = PaddleMotor->STS.Idle && Shooter->STS.Disabled;
	BallControl->STS.AutoActive = PaddleMotor->STS.AutoActive && Shooter->STS.AutoActive;
	BallControl->STS.Disabled = PaddleMotor->STS.Disabled && Shooter->STS.Disabled;
	BallControl->STS.Initializing = PaddleMotor->STS.Initializing && Shooter->STS.Disabled;
	BallControl->STS.Running = PaddleMotor->STS.Running && (Shooter->STS.Idle || Shooter->STS.Shooting);
	BallControl->STS.Interlocked = PaddleMotor->STS.Interlocked || Shooter->STS.Interlocked;

	/* any subsystem alarm */
	BOOL sensorAlarm = DistanceSensorLeft->STS.AlarmActive || DistanceSensorMiddle->STS.AlarmActive || DistanceSensorRight->STS.AlarmActive;
	BallControl->STS.AlarmActive = PaddleMotor->STS.AlarmActive || Shooter->STS.AlarmActive || sensorAlarm;

}
```

#### FB_FieldControl.c
```c
/*********************************************************************************
 * Copyright: MyAutomation-IT
 * Author:    raivo
 * Created:   April 22, 2026/5:57 PM
 *********************************************************************************/
#include <bur/plctypes.h>
#include "CommonTypes.h"
#ifdef __cplusplus
	extern "C"
	{
#endif
	#include "Library.h"
#ifdef __cplusplus
	};
#endif

#define MAX_ANGLE 18
#define MIN_ANGLE 3

#define FieldMotor inst->FieldMotor
#define FieldControl inst->FieldControl
#define InclinoSensor inst->InclinoSensor

#define STOPPING_OFFSET (FieldControl->PAR.Angle * -0.068) + 1.3

/* TODO: Add your comment here */
void FB_FieldControl(struct FB_FieldControl* inst)
{

	if(FieldControl->CS.StopGame)
	{
		FieldControl->STS.StateInt = STATE_STOPPING;
	}

	switch(FieldControl->STS.StateInt)
	{
		case STATE_DISABLED:
		{
			FieldControl->STS.AtTargetPosition = 0;

			if(FieldControl->HMI.IncreaseAngle && FieldControl->PAR.Angle < MAX_ANGLE)
			{
				FieldControl->PAR.Angle += 0.002;
			}
			else if(FieldControl->HMI.DecreaseAngle && FieldControl->PAR.Angle > MIN_ANGLE)
			{
				FieldControl->PAR.Angle -= 0.002;
			}
			if(FieldControl->STS.Initializing)
			{
				FieldControl->STS.StateInt = STATE_INITIALIZING;
			}
			break;
		}
		case STATE_INITIALIZING:
		{
			if(FieldControl->STS.Idle)
			{
				FieldControl->STS.StateInt = STATE_IDLE;
			}
			else if((FieldControl->STS.CurrentAngle + STOPPING_OFFSET >= FieldControl->PAR.Angle) && !FieldControl->STS.AtTargetPosition && FieldMotor->STS.EndButtonHit)
			{
				FieldControl->STS.AtTargetPosition = 1;
			}
			break;
		}
		case STATE_IDLE:
		{
			if(FieldControl->STS.Running)
			{
				FieldControl->STS.StateInt = STATE_RUNNING;
			}
			break;
		}
		case STATE_RUNNING:
		{
			FieldMotor->CS.Stop = 0;
			if(FieldControl->STS.CurrentAngle >= MAX_ANGLE)
			{
				FieldMotor->HMI.MoveJogNeg = 0;
			}
			break;
		}
		case STATE_STOPPING:
		{
			if(FieldControl->STS.Disabled)
			{
				FieldControl->STS.StateInt = STATE_DISABLED;
			}
			break;
		}
	}

	/*TODO: Add your code here*/
	FieldMotor->CS.Initialize = FieldControl->CS.Initialize;
	FieldMotor->CS.Start = FieldControl->CS.Start;
	FieldMotor->CS.StopGame = FieldControl->CS.StopGame;
	FieldMotor->CS.ErrorAcknowledge = FieldControl->CS.ErrorAcknowledge;
	FieldMotor->STS.AtTargetPosition = FieldControl->STS.AtTargetPosition;

	FieldControl->STS.CurrentAngle = InclinoSensor->STS.CurrentAngle;
	FieldControl->STS.Disabled = FieldMotor->STS.Disabled;
	FieldControl->STS.AlarmActive = FieldMotor->STS.AlarmActive || InclinoSensor->STS.AlarmActive;
	FieldControl->STS.Interlocked = FieldMotor->STS.Interlocked;
	FieldControl->STS.Idle = FieldMotor->STS.Idle;
	FieldControl->STS.Running = FieldMotor->STS.Running;
	FieldControl->STS.Moving = FieldMotor->STS.Moving;
	FieldControl->STS.Initializing = FieldMotor->STS.Initializing;

	FieldControl->CS.SetCenterPoint = FieldMotor->CS.SetCenterPoint;
	InclinoSensor->CS.SetCenterPoint = FieldMotor->CS.SetCenterPoint;

}
```

#### FB_PongGame.c
```c
/*********************************************************************************
 * Copyright: MyAutomation-IT
 * Author:    raivo
 * Created:   April 22, 2026/5:57 PM
 *********************************************************************************/
#include <bur/plctypes.h>
#include <standard.h>
#include "CommonTypes.h"
#ifdef __cplusplus
	extern "C"
	{
#endif
	#include "Library.h"
#ifdef __cplusplus
	};
#endif

#define PongGame inst->PongGame
#define BallControl inst->BallControl
#define FieldControl inst->FieldControl

_LOCAL TON_typ AlarmTimer;
_LOCAL BOOL BlinkState;

/* TODO: Add your comment here */
void FB_PongGame(struct FB_PongGame* inst)
{
	if(PongGame->CS.StopGame || PongGame->HMI.StopGame)
	{
		PongGame->STS.StateInt = STATE_STOPPING;
	}
	PongGame->STS.AlarmActiveColour = BLACK_COLOUR;
	if(PongGame->STS.AlarmActive)
	{
		PongGame->CS.StopGame = !PongGame->STS.GameStopped;

		if(PongGame->CS.StopGame && !PongGame->STS.GameStopped)
		{
    		PongGame->STS.GameStopped = 1;
			//PongGame->CS.StopGame = 0;
		}

		AlarmTimer.IN = 1;
		AlarmTimer.PT = 1000;
		TON(&AlarmTimer);

		if(AlarmTimer.Q)
		{
			BlinkState = !BlinkState;

			AlarmTimer.IN = 0;
			TON(&AlarmTimer);
		}
		if(BlinkState)
		{
			PongGame->STS.AlarmActiveColour = RED_COLOUR;
		}
		else
		{
			PongGame->STS.AlarmActiveColour = BLACK_COLOUR;
		}
	}
	else
	{
		AlarmTimer.IN = 0;
		TON(&AlarmTimer);
		BlinkState = 0;
	}

	switch(PongGame->STS.StateInt)
	{
		case STATE_DISABLED:
		{
			PongGame->STS.GameStopped = 0;
			PongGame->CS.StopGame = 0;
			strncpy(PongGame->STS.StateString, "Disabled", sizeof(PongGame->STS.StateString));
			if(PongGame->STS.Initializing)
			{
				PongGame->STS.StateInt = STATE_INITIALIZING;
			}
			break;
		}
		case STATE_INITIALIZING:
		{
			strncpy(PongGame->STS.StateString, "Initializing...", sizeof(PongGame->STS.StateString));
			if(PongGame->STS.Idle)
			{
				PongGame->STS.StateInt = STATE_IDLE;
			}
			break;
		}
		case STATE_IDLE:
		{
			strncpy(PongGame->STS.StateString, "Idle", sizeof(PongGame->STS.StateString));
			if(PongGame->STS.Running)
			{
				PongGame->STS.StateInt = STATE_RUNNING;
			}
			break;
		}
		case STATE_RUNNING:
		{
			strncpy(PongGame->STS.StateString, "Running", sizeof(PongGame->STS.StateString));
			break;
		}
		case STATE_STOPPING:
		{
			strncpy(PongGame->STS.StateString, "Stopping...", sizeof(PongGame->STS.StateString));
			if(PongGame->STS.Disabled)
			{
				PongGame->STS.StateInt = STATE_DISABLED;
			}
			break;
		}
	}

	BallControl->CS.Initialize = PongGame->HMI.Initialize ^ PongGame->CS.Initialize;
	BallControl->CS.StopGame = PongGame->HMI.StopGame ^ PongGame->CS.StopGame;
	BallControl->CS.Start = PongGame->HMI.Start ^ PongGame->CS.Start;
	BallControl->CS.AutoMode = PongGame->HMI.AutoMode ^ PongGame->CS.AutoMode;
	BallControl->CS.ErrorAcknowledge = PongGame->HMI.ErrorAcknowledge ^ PongGame->CS.ErrorAcknowledge;

	FieldControl->CS.Initialize = PongGame->HMI.Initialize ^ PongGame->CS.Initialize;
	FieldControl->CS.StopGame = PongGame->HMI.StopGame ^ PongGame->CS.StopGame;
	FieldControl->CS.Start = PongGame->HMI.Start ^ PongGame->CS.Start;

	FieldControl->STS.AutoActive = PongGame->HMI.AutoMode || PongGame->CS.AutoMode;

	PongGame->STS.AutoActive = BallControl->STS.AutoActive && FieldControl->STS.AutoActive;
	PongGame->STS.Initializing = BallControl->STS.Initializing && FieldControl->STS.Initializing;
	PongGame->STS.AlarmActive = BallControl->STS.AlarmActive || FieldControl->STS.AlarmActive;
	PongGame->STS.Disabled = BallControl->STS.Disabled && FieldControl->STS.Disabled;
	PongGame->STS.Idle = BallControl->STS.Idle && FieldControl->STS.Idle;
	PongGame->STS.Running = BallControl->STS.Running && FieldControl->STS.Running;
	PongGame->STS.Interlocked = BallControl->STS.Interlocked || FieldControl->STS.Interlocked;
}
```

#### CommonTypes.h
```c
/*********************************************************************************
 * Copyright: MyAutomation-IT
 * Author:    raivo
 * Created:   April 22, 2026/5:57 PM
 *********************************************************************************/
#ifndef COMMON_TYPES_H
#define COMMON_TYPES_H

#define ENDBUTTON_BITMASK_FIELD 0x4
#define ENDBUTTON_BITMASK_PADDLE 0x2

#define TO_DEGREES 100
#define SHIFT_BYTE 8

#define CENTERPOINT_NORMAL 7
#define CENTERPOINT_SET 3

#define BLACK_COLOUR 0
#define GREEN_COLOUR 10
#define RED_COLOUR   51

#define STATE_DISABLED 0
#define STATE_INITIALIZING 10
#define STATE_IDLE 20
#define STATE_RUNNING 30
#define STATE_STOPPING 40

#define STATE_SHOOTING 30
#define SHOOT_OUTPUT_BIT 3
#define FAN_OUTPUT_BIT 0

#define MS_50 50
#define MS_100 100
#define MS_500 500
#define MS_1000 1000

#define MAX_ACC_DEC 40000
#define MAX_VELOCITY 2000
#define MIN_VELOCITY 100
#define STD_VELOCITY 1000
#define MIN_POSITION (PaddleMotor->STS.ReferencePosition - MAX_PADDLE_DISTANCE_TICKS)

#define OVERLOAD 32760
#define UNDERLOAD -32760
#define SHIFT_BYTE 8
#define NUM_SENSORS 3

#define OUT1_BITMASK 0x1
#define OUT2_BITMASK 0x2
#define DEVICE_STATUS_BITMASK 0xF0
#define SENSOR_FAILURE 4

#define BALL_MIN_DISTANCE 50
#define BALL_MAX_DISTANCE 300

#define MM_TO_POSITION 11.2
#define MAX_POSITION (PaddleMotor->STS.ReferencePosition - 100)
#define AUTOMODE_VELOCITY 5000
#define MIN_FIELD_DISTANCE 50
#define MAX_INTENSITY 10
#define MIN_INTENSITY 3

#define MAX_ANGLE 18
#define MIN_ANGLE 3

#define DISTANCE_BETWEEN_SENSORS_MM 24
#define DISTANCE_SENSOR_LEFT_TO_PADDLE_MM 75

#define GAME_OVER_TRIGGER_MS 5000

static const float MAX_PADDLE_DISTANCE_MM = 222.0f;
static const float MAX_PADDLE_DISTANCE_TICKS = 2830.0f;

static const float TICKS_TO_MM = 222.0f / 2830.0f;
static const float MM_TO_TICKS = 2830.0f / 222.0f;
#endif
```

#### ActPositionToMM.c - not listed in the package file held
```c
#include <bur/plctypes.h>
#ifdef __cplusplus
	extern "C"
	{
#endif
	#include "Library.h"
#ifdef __cplusplus
	};
#endif

	/*TODO: Add your code here*/
#define ACTPOSITION_TO_MM 0.0784

/* TODO: Add your comment here */
unsigned short ActPositionToMM(float ActPosition)
{
	return (UINT)((-ActPosition) * ACTPOSITION_TO_MM);
}

unsigned char SetOutputs(unsigned char digitalOutputs, plcbit ventilator, plcbit solenoid)
{
	digitalOutputs &= ~((1 << 0) | (1 << 3));
	digitalOutputs |= ((USINT)ventilator << 0) | ((USINT)solenoid << 3);

	return digitalOutputs;
}

short SensorDataConverter(unsigned char MSB, unsigned char LSB)
{
	return (INT)((MSB << 8) | LSB);
}

float InclineSensorDataToAngle(INT InclineSensorData)
{
	return (float)(InclineSensorData) / 100;
}
```

### Program Logical/Libraries/Timer

#### IECTimerFactory.hpp
```cpp
/********************************************************************
 * COPYRIGHT --
 ********************************************************************
 * Library: Timer
 * File: IECTimerFactory.hpp
 *******************************************************************/
#pragma once

#include "IECTonTimer.hpp"
#include "IECTofTimer.hpp"
#include "IECTpTimer.hpp"

/* Concrete factory for IEC timer */
class IECTimerFactory : public TimerFactory
{
	public:
		IECTimerFactory() {};

		virtual ~IECTimerFactory(){};

		virtual ITimer* createTON(signed long time = 0) const
		{
			return new IECTonTimer(time);
		}

		virtual ITimer* createTOF(signed long time = 0) const
		{
			return new IECTofTimer(time);
		}

		virtual ITimer* createTP(signed long time = 0)  const
		{
			return new IECTpTimer(time);
		}

		static TimerFactory* getInstance();
};
```

#### IECTpTimer.hpp
```cpp
/********************************************************************
 * COPYRIGHT --
 ********************************************************************
 * Library: Timer
 * File: IECTonTimer.hpp
 *******************************************************************/
#pragma once

#include <standard.h>
#include "ITimer.hpp"

/* The class IECTonTimer wraps a B&R TP (pulse generator) function block.
*/
class IECTpTimer : public ITimer
{
	private:
		TP_typ fubTP;

	public:
		IECTpTimer();
		IECTpTimer(signed long time);
		virtual ~IECTpTimer() {};
		virtual void start(bool start = 1);
		virtual void reset(bool reset = 1);
		virtual bool output();
		virtual void setTime(signed long time);
		virtual signed long getElapsedTime();

		virtual void cyclic();
};
```

#### ITimer.hpp
```cpp
/********************************************************************
 * COPYRIGHT --
 ********************************************************************
 * Library: Timer
 * File: ITimer.hpp
 *******************************************************************/
#pragma once

/* Interface timer class */
class ITimer
{
	public:
		ITimer() {};
		ITimer(signed long time);
		virtual ~ITimer() {};
		virtual void start(bool start = 1) = 0;
		virtual void reset(bool reset = 1) = 0;
		virtual bool output() = 0;
		virtual void setTime(signed long time) = 0;
		virtual signed long getElapsedTime() = 0;
		virtual void cyclic() = 0;
};

/* Superclass for concrete timer factory classes */
class TimerFactory
{
	public:
		TimerFactory() {};
		virtual ~TimerFactory(){};
		virtual ITimer* createTON(signed long time = 0) const = 0;
		virtual ITimer* createTOF(signed long time = 0) const = 0;
		virtual ITimer* createTP(signed long time = 0)  const = 0;
		static TimerFactory* getInstance();
};
```

#### Timer.hpp
```cpp
/********************************************************************
 * COPYRIGHT --
 ********************************************************************
 * Library: Timer
 * File: Timer.hpp
 *******************************************************************/
#pragma once

#include "ITimer.hpp"
#include "IECTonTimer.hpp"
#include "IECTofTimer.hpp"
#include "IECTpTimer.hpp"
```

#### IECTimerFactory.cpp
```cpp
/********************************************************************
 * COPYRIGHT --
 ********************************************************************
 * Library: Timer
 * File: IECTimerFactory.cpp
 *******************************************************************/

#include "ITimer.hpp"
#include "IECTimerFactory.hpp"

/* Create a concrete IEC factory */
TimerFactory* TimerFactory::getInstance()
{
	static IECTimerFactory theIECTimerFactory;
	return &theIECTimerFactory;
}
```

#### IECTofTimer.cpp
```cpp
/********************************************************************
 * COPYRIGHT --
 ********************************************************************
 * Library: Timer
 * File: IECTofTimer.cpp
 *******************************************************************/

#include <bur/plctypes.h>
#include <string.h>
#include "IECTofTimer.hpp"

IECTofTimer::IECTofTimer()
{
	memset(&fubTOF,0,sizeof(fubTOF));
}

IECTofTimer::IECTofTimer(signed long time)
{
	memset(&fubTOF,0,sizeof(fubTOF));
	this->setTime(time);
}

void IECTofTimer::start(bool start)
{
	this->fubTOF.IN = start;
}

void IECTofTimer::reset(bool reset)
{
	this->fubTOF.IN = !reset;
}

void IECTofTimer::setTime(signed long time)
{
	this->fubTOF.PT = time;
}

bool IECTofTimer::output()
{
	return this->fubTOF.Q;
}

signed long IECTofTimer::getElapsedTime()
{
	return this->fubTOF.ET;
}

/* This method has to be called cyclically in programms. */
void IECTofTimer::cyclic()
{
	TOF(&fubTOF);
}
```

#### IECTonTimer.cpp
```cpp
/********************************************************************
 * COPYRIGHT --
 ********************************************************************
 * Library: Timer
 * File: IECTonTimer.cpp
 *******************************************************************/

#include <bur/plctypes.h>
#include <string.h>
#include "IECTonTimer.hpp"

IECTonTimer::IECTonTimer()
{
	memset(&fubTON,0,sizeof(fubTON));
}

IECTonTimer::IECTonTimer(signed long time)
{
	memset(&fubTON,0,sizeof(fubTON));
	this->setTime(time);
}

void IECTonTimer::start(bool start)
{
	this->fubTON.IN = start;
}

void IECTonTimer::reset(bool reset)
{
	this->fubTON.IN = !reset;
}

void IECTonTimer::setTime(signed long time)
{
	this->fubTON.PT = time;
}

bool IECTonTimer::output()
{
	return this->fubTON.Q;
}

signed long IECTonTimer::getElapsedTime()
{
	return this->fubTON.ET;
}

/* This method has to be called cyclically in programms. */
void IECTonTimer::cyclic()
{
	TON(&fubTON);
}
```

- Visualisation Logical/mappView (not shown)

### Program Logical/Main (ANSIC)

#### Cyclic.cpp - Cyclic code
```cpp
#include <bur/plctypes.h>
#ifdef _DEFAULT_INCLUDES
	#include <AsDefault.h>
#endif

// amount of memory to be allocated for heap storage must be specified for every ANSI C++ program with the bur_heap_size variable
unsigned long bur_heap_size = 0xFFFF;

void _CYCLIC ProgramCyclic(void)
{
	PaddleMotor.digitalInput = digitalInput;
	FieldMotor.digitalInput = digitalInput;

	FB_PaddleMotor(&PaddleMotor);
	FB_Shooter(&Shooter);
	FB_DistanceSensor(&DistanceSensors);
	FB_FieldMotor(&FieldMotor);
	FB_InclinoSensor(&InclinoSensor);
	FB_FieldControl(&FieldControl);
	FB_BallControl(&BallControl);
	FB_PongGame(&PongGame);

	digitalOutput = Shooter.digitalOutput;

	if(g_PongGame.PAR.Highscore > g_Highscore)
	{
		g_Highscore = g_PongGame.PAR.Highscore;
	}
}
```

#### Init.cpp - Initialization code
```cpp
#include <bur/plctypes.h>

#ifdef _DEFAULT_INCLUDES
	#include <AsDefault.h>
#endif

void _INIT ProgramInit(void)
{

	g_PaddleMotor.PAR.Velocity = 1000;
	g_PaddleMotor.PAR.Acceleration = 5000;
	g_PaddleMotor.PAR.Deceleration = 5000;
	g_PaddleMotor.PAR.JogVelocity = 400;

	g_FieldMotor.PAR.Velocity = 1000;
	g_FieldMotor.PAR.Acceleration = 5000;
	g_FieldMotor.PAR.Deceleration = 5000;
	g_FieldMotor.PAR.JogVelocity = 400;
}
```

#### Variables.var - Local variables
```iecst
VAR
	DistanceSensors : FB_DistanceSensor;
	PaddleMotor : FB_PaddleMotor;
	Shooter : FB_Shooter;
	InclinoSensor : FB_InclinoSensor;
	FieldMotor : FB_FieldMotor;
	FieldControl : FB_FieldControl;
	BallControl : FB_BallControl;
	PongGame : FB_PongGame;
END_VAR
```

### Data object Logical/acp10etxen (Ett)

- acp10etxen.ett (not shown)

### Package Logical/gAxis01obj - gAxis01obj

### Program Logical/gAxis01obj/gAxis01Basic (ANSIC) - Basic logical control

#### basic.typ
```iecst
TYPE
	basic_command_typ : 	STRUCT  (*command structure*)
		Power : BOOL; (*switch on the controller*)
		Home : BOOL; (*reference the axis*)
		MoveAbsolute : BOOL; (*move to an defined position*)
		MoveAdditive : BOOL; (*move a defiened distance*)
		MoveVelocity : BOOL; (*start a movement with a defiened velocity*)
		Halt : BOOL; (*stop every active movement once*)
		Stop : BOOL; (*stop every active movement as long as set*)
		MoveJogPos : BOOL; (*move in positive direction as long as is set*)
		MoveJogNeg : BOOL; (*move in negative direction as long as is set*)
		ErrorAcknowledge : BOOL; (*reset active errors*)
	END_STRUCT;
	basic_parameter_typ : 	STRUCT  (*parameter structure*)
		Position : REAL; (*target-position for MoveAbsolute-Command*)
		Distance : REAL; (*distance for MoveAdditive-Command*)
		Velocity : REAL; (*velocity for MoveVelocity-Command*)
		Direction : USINT; (*direction for commanded movements*)
		Acceleration : REAL; (*acceleration for commanded movements*)
		Deceleration : REAL; (*deceleration for commanded movements*)
		HomePosition : REAL; (*target-position for referencing the axis*)
		HomeMode : USINT; (*homing mode*)
		JogVelocity : REAL; (*velocity for jogging movement*)
	END_STRUCT;
	basic_status_typ : 	STRUCT  (*status structure*)
		ErrorID : UINT; (*ErrorID of any occured error*)
		ErrorText : ARRAY[0..3]OF STRING[79]; (*Error Text*)
		ActPosition : REAL; (*actual position of the axis*)
		ActVelocity : REAL; (*actual velocity of the axis*)
		DriveStatus : MC_DRIVESTATUS_TYP; (*actual status of the axis*)
	END_STRUCT;
	basic_axisState_typ : 	STRUCT  (*axis state structure*)
		Disabled : BOOL; (*if set, axis is in state Disabled*)
		StandStill : BOOL; (*if set, axis is in state StandsStill*)
		Homing : BOOL; (*if set, axis is in state Homing*)
		Stopping : BOOL; (*if set, axis is in state Stopping*)
		DiscreteMotion : BOOL; (*if set, axis is in state DiscreteMotion*)
		ContinuousMotion : BOOL; (*if set, axis is in state ContinuousMotion*)
		SynchronizedMotion : BOOL; (*if set, axis is in state SynchronizedMotion*)
		ErrorStop : BOOL; (*if set, axis is in state ErrorStop*)
	END_STRUCT;
	basic_typ : 	STRUCT  (*control structure*)
		Command : basic_command_typ; (*command structure*)
		Parameter : basic_parameter_typ; (*parameter structure*)
		Status : basic_status_typ; (*status structure*)
		AxisState : basic_axisState_typ; (*axis state structure*)
	END_STRUCT;
END_TYPE
```

#### basic.var
```iecst
VAR
	BasicControl : basic_typ; (*control structure*)
	MC_BR_ReadDriveStatus_0 : MC_BR_ReadDriveStatus; (*Function Block*)
	MC_Halt_0 : MC_Halt; (*Function Block*)
	MC_Home_0 : MC_Home; (*Function Block*)
	MC_MoveAbsolute_0 : MC_MoveAbsolute; (*Function Block*)
	MC_MoveAdditive_0 : MC_MoveAdditive; (*Function Block*)
	MC_MoveVelocity_0 : MC_MoveVelocity; (*Function Block*)
	MC_Power_0 : MC_Power; (*Function Block*)
	MC_ReadActualPosition_0 : MC_ReadActualPosition; (*Function Block*)
	MC_ReadActualVelocity_0 : MC_ReadActualVelocity; (*Function Block*)
	MC_ReadAxisError_0 : MC_ReadAxisError; (*Function Block*)
	MC_ReadStatus_0 : MC_ReadStatus; (*Function Block*)
	MC_Reset_0 : MC_Reset; (*Function Block*)
	MC_Stop_0 : MC_Stop; (*Function Block*)
	Axis1Obj : UDINT; (*axis reference*)
	AxisStep : USINT;
END_VAR
```
